LIN {X 0,Y 302.598,Z 692.488,A -85,B 0,C 180,E1 10469.522,E2 10469.522} C_VEL
LIN {X 0,Y 304.886,Z 667.23,A -85,B 0,C 180,E1 10468.838,E2 10468.838} C_VEL
LIN {X 0,Y 315.43,Z 536.888,A -85,B 0,C 180,E1 10466.199,E2 10466.199} C_VEL
LIN {X 0,Y 309.663,Z 526.865,A -85,B 0,C 180,E1 10462.898,E2 10462.898} C_VEL
LIN {X 0,Y 304.796,Z 519.088,A -85,B 0,C 180,E1 10459.549,E2 10459.549} C_VEL
LIN {X 0,Y 301.581,Z 514.357,A -85,B 0,C 180,E1 10456.864,E2 10456.864} C_VEL
LIN {X 0,Y 300.41,Z 512.771,A -85,B 0,C 180,E1 10455.75,E2 10455.75} C_VEL
LIN {X 0,Y 298.97,Z 511.709,A -85,B 0,C 180,E1 10454.313,E2 10454.313} C_VEL
LIN {X 0,Y 296.741,Z 512.653,A -85,B 0,C 180,E1 10451.996,E2 10451.996} C_VEL
LIN {X 0,Y 294.887,Z 513.836,A -85,B 0,C 180,E1 10449.52,E2 10449.52} C_VEL
LIN {X 0,Y 294.603,Z 513.741,A -85,B 0,C 180,E1 10448.976,E2 10448.976} C_VEL
LIN {X 0,Y 293.288,Z 512.887,A -85,B 0,C 180,E1 10444.302,E2 10444.302} C_VEL
LIN {X 0,Y 293.492,Z 513.574,A -85,B 0,C 180,E1 10440.391,E2 10440.391} C_VEL
LIN {X 0,Y 295.393,Z 518.005,A -85,B 0,C 180,E1 10435.341,E2 10435.341} C_VEL
LIN {X 0,Y 297.878,Z 523.02,A -85,B 0,C 180,E1 10431.799,E2 10431.799} C_VEL
LIN {X 0,Y 299.981,Z 527.143,A -85,B 0,C 180,E1 10429.534,E2 10429.534} C_VEL
LIN {X 0,Y 303.204,Z 533.381,A -85,B 0,C 180,E1 10426.703,E2 10426.703} C_VEL
LIN {X 0,Y 307.026,Z 541.211,A -85,B 0,C 180,E1 10423.882,E2 10423.882} C_VEL
LIN {X 0,Y 311.626,Z 551.031,A -85,B 0,C 180,E1 10420.995,E2 10420.995} C_VEL
LIN {X 0,Y 312.497,Z 553.268,A -85,B 0,C 180,E1 10420.473,E2 10420.473} C_VEL
LIN {X 0,Y 297.53,Z 720.46,A -85,B 0,C 180,E1 10416.945,E2 10416.945} C_VEL
LIN {X 0,Y 293.952,Z 742.565,A -85,B 0,C 180,E1 10416.298,E2 10416.298} C_VEL
LIN {X 0,Y 288.986,Z 764.025,A -85,B 0,C 180,E1 10415.487,E2 10415.487} C_VEL
LIN {X 0,Y 282.983,Z 784.23,A -85,B 0,C 180,E1 10414.512,E2 10414.512} C_VEL
LIN {X 0,Y 275.952,Z 803.851,A -85,B 0,C 180,E1 10413.261,E2 10413.261} C_VEL
LIN {X 0,Y 268.029,Z 822.907,A -85,B 0,C 180,E1 10411.679,E2 10411.679} C_VEL
LIN {X 0,Y 258.872,Z 842.398,A -85,B 0,C 180,E1 10409.605,E2 10409.605} C_VEL
LIN {X 0,Y 249.5,Z 860.393,A -85,B 0,C 180,E1 10407.16,E2 10407.16} C_VEL
LIN {X 0,Y 239.675,Z 877.621,A -85,B 0,C 180,E1 10404.172,E2 10404.172} C_VEL
LIN {X 0,Y 230.079,Z 893.458,A -85,B 0,C 180,E1 10400.667,E2 10400.667} C_VEL
LIN {X 0,Y 220.636,Z 908.459,A -85,B 0,C 180,E1 10396.464,E2 10396.464} C_VEL
LIN {X 0,Y 212.557,Z 921.328,A -85,B 0,C 180,E1 10391.906,E2 10391.906} C_VEL
LIN {X 0,Y 205.237,Z 933.456,A -85,B 0,C 180,E1 10386.463,E2 10386.463} C_VEL
LIN {X 0,Y 199.633,Z 943.745,A -85,B 0,C 180,E1 10380.521,E2 10380.521} C_VEL
LIN {X 0,Y 196.02,Z 952.022,A -85,B 0,C 180,E1 10374.402,E2 10374.402} C_VEL
LIN {X 0,Y 194.187,Z 958.687,A -85,B 0,C 180,E1 10367.994,E2 10367.994} C_VEL
LIN {X 0,Y 193.926,Z 963.068,A -85,B 0,C 180,E1 10362.204,E2 10362.204} C_VEL
LIN {X 0,Y 194.453,Z 965.803,A -85,B 0,C 180,E1 10356.792,E2 10356.792} C_VEL
LIN {X 0,Y 194.986,Z 966.923,A -85,B 0,C 180,E1 10352.352,E2 10352.352} C_VEL
LIN {X 0,Y 195.041,Z 967.009,A -85,B 0,C 180,E1 10348.457,E2 10348.457} C_VEL
LIN {X 0,Y 194.615,Z 966.173,A -85,B 0,C 180,E1 10344.4,E2 10344.4} C_VEL
LIN {X 0,Y 194.022,Z 963.972,A -85,B 0,C 180,E1 10339.311,E2 10339.311} C_VEL
LIN {X 0,Y 194.046,Z 959.689,A -85,B 0,C 180,E1 10333.232,E2 10333.232} C_VEL
LIN {X 0,Y 195.44,Z 953.707,A -85,B 0,C 180,E1 10327.051,E2 10327.051} C_VEL
LIN {X 0,Y 198.684,Z 945.671,A -85,B 0,C 180,E1 10320.786,E2 10320.786} C_VEL
LIN {X 0,Y 203.684,Z 936.028,A -85,B 0,C 180,E1 10314.952,E2 10314.952} C_VEL
LIN {X 0,Y 210.542,Z 924.446,A -85,B 0,C 180,E1 10309.419,E2 10309.419} C_VEL
LIN {X 0,Y 218.263,Z 912.191,A -85,B 0,C 180,E1 10304.768,E2 10304.768} C_VEL
LIN {X 0,Y 227.319,Z 897.792,A -85,B 0,C 180,E1 10300.461,E2 10300.461} C_VEL
LIN {X 0,Y 236.604,Z 882.589,A -85,B 0,C 180,E1 10296.875,E2 10296.875} C_VEL
LIN {X 0,Y 246.735,Z 865.128,A -85,B 0,C 180,E1 10293.627,E2 10293.627} C_VEL
LIN {X 0,Y 256.161,Z 847.562,A -85,B 0,C 180,E1 10291.056,E2 10291.056} C_VEL
LIN {X 0,Y 265.436,Z 828.501,A -85,B 0,C 180,E1 10288.873,E2 10288.873} C_VEL
LIN {X 0,Y 273.54,Z 809.538,A -85,B 0,C 180,E1 10287.187,E2 10287.187} C_VEL
LIN {X 0,Y 280.979,Z 789.632,A -85,B 0,C 180,E1 10285.817,E2 10285.817} C_VEL
LIN {X 0,Y 287.475,Z 769.122,A -85,B 0,C 180,E1 10284.747,E2 10284.747} C_VEL
LIN {X 0,Y 293.011,Z 746.686,A -85,B 0,C 180,E1 10283.853,E2 10283.853} C_VEL
LIN {X 0,Y 296.814,Z 724.483,A -85,B 0,C 180,E1 10283.178,E2 10283.178} C_VEL
LIN {X 0,Y 299.999,Z 692.914,A -85,B 0,C 180,E1 10282.46,E2 10282.46} C_VEL
LIN {X 0,Y 312.304,Z 552.77,A -85,B 0,C 180,E1 10279.497,E2 10279.497} C_VEL
LIN {X 0,Y 307.54,Z 542.415,A -85,B 0,C 180,E1 10276.576,E2 10276.576} C_VEL
LIN {X 0,Y 303.48,Z 534.184,A -85,B 0,C 180,E1 10273.673,E2 10273.673} C_VEL
LIN {X 0,Y 300.18,Z 527.74,A -85,B 0,C 180,E1 10270.847,E2 10270.847} C_VEL
LIN {X 0,Y 298.085,Z 523.643,A -85,B 0,C 180,E1 10268.681,E2 10268.681} C_VEL
LIN {X 0,Y 296.396,Z 520.441,A -85,B 0,C 180,E1 10266.586,E2 10266.586} C_VEL
LIN {X 0,Y 294.859,Z 517.125,A -85,B 0,C 180,E1 10264.083,E2 10264.083} C_VEL
LIN {X 0,Y 293.192,Z 513.211,A -85,B 0,C 180,E1 10259.218,E2 10259.218} C_VEL
LIN {X 0,Y 293.326,Z 512.761,A -85,B 0,C 180,E1 10253.934,E2 10253.934} C_VEL
LIN {X 0,Y 294.723,Z 513.985,A -85,B 0,C 180,E1 10250.233,E2 10250.233} C_VEL
LIN {X 0,Y 298.119,Z 518.939,A -85,B 0,C 180,E1 10245.332,E2 10245.332} C_VEL
LIN {X 0,Y 301.263,Z 523.806,A -85,B 0,C 180,E1 10242.221,E2 10242.221} C_VEL
LIN {X 0,Y 304.449,Z 528.849,A -85,B 0,C 180,E1 10239.677,E2 10239.677} C_VEL
LIN {X 0,Y 309.247,Z 536.938,A -85,B 0,C 180,E1 10236.465,E2 10236.465} C_VEL
LIN {X 0,Y 311.824,Z 541.761,A -85,B 0,C 180,E1 10234.936,E2 10234.936} C_VEL
LIN {X 0,Y 300.184,Z 680.951,A -85,B 0,C 180,E1 10232.1,E2 10232.1} C_VEL
LIN {X 0,Y 297.715,Z 701.831,A -85,B 0,C 180,E1 10231.431,E2 10231.431} C_VEL
LIN {X 0,Y 293.977,Z 722.266,A -85,B 0,C 180,E1 10230.528,E2 10230.528} C_VEL
LIN {X 0,Y 289.19,Z 741.453,A -85,B 0,C 180,E1 10229.407,E2 10229.407} C_VEL
LIN {X 0,Y 283.05,Z 761.038,A -85,B 0,C 180,E1 10227.961,E2 10227.961} C_VEL
LIN {X 0,Y 275.997,Z 779.593,A -85,B 0,C 180,E1 10226.234,E2 10226.234} C_VEL
LIN {X 0,Y 268.131,Z 797.188,A -85,B 0,C 180,E1 10224.19,E2 10224.19} C_VEL
LIN {X 0,Y 259.42,Z 813.987,A -85,B 0,C 180,E1 10221.736,E2 10221.736} C_VEL
LIN {X 0,Y 250.527,Z 829.117,A -85,B 0,C 180,E1 10218.957,E2 10218.957} C_VEL
LIN {X 0,Y 241.45,Z 843.036,A -85,B 0,C 180,E1 10215.751,E2 10215.751} C_VEL
LIN {X 0,Y 232.571,Z 855.538,A -85,B 0,C 180,E1 10212.112,E2 10212.112} C_VEL
LIN {X 0,Y 224.082,Z 866.647,A -85,B 0,C 180,E1 10208.001,E2 10208.001} C_VEL
LIN {X 0,Y 215.89,Z 876.71,A -85,B 0,C 180,E1 10203.122,E2 10203.122} C_VEL
LIN {X 0,Y 209.066,Z 884.767,A -85,B 0,C 180,E1 10197.945,E2 10197.945} C_VEL
LIN {X 0,Y 203.512,Z 891.329,A -85,B 0,C 180,E1 10192.225,E2 10192.225} C_VEL
LIN {X 0,Y 199.383,Z 896.318,A -85,B 0,C 180,E1 10186.008,E2 10186.008} C_VEL
LIN {X 0,Y 197.027,Z 899.441,A -85,B 0,C 180,E1 10179.934,E2 10179.934} C_VEL
LIN {X 0,Y 195.894,Z 901.059,A -85,B 0,C 180,E1 10173.803,E2 10173.803} C_VEL
LIN {X 0,Y 195.752,Z 901.224,A -85,B 0,C 180,E1 10167.95,E2 10167.95} C_VEL
LIN {X 0,Y 196.557,Z 900.078,A -85,B 0,C 180,E1 10161.811,E2 10161.811} C_VEL
LIN {X 0,Y 198.545,Z 897.495,A -85,B 0,C 180,E1 10155.715,E2 10155.715} C_VEL
LIN {X 0,Y 202.162,Z 893.041,A -85,B 0,C 180,E1 10149.443,E2 10149.443} C_VEL
LIN {X 0,Y 207.241,Z 887,A -85,B 0,C 180,E1 10143.651,E2 10143.651} C_VEL
LIN {X 0,Y 213.604,Z 879.489,A -85,B 0,C 180,E1 10138.384,E2 10138.384} C_VEL
LIN {X 0,Y 221.371,Z 870.076,A -85,B 0,C 180,E1 10133.405,E2 10133.405} C_VEL
LIN {X 0,Y 229.529,Z 859.758,A -85,B 0,C 180,E1 10129.204,E2 10129.204} C_VEL
LIN {X 0,Y 238.649,Z 847.341,A -85,B 0,C 180,E1 10125.267,E2 10125.267} C_VEL
LIN {X 0,Y 247.506,Z 834.121,A -85,B 0,C 180,E1 10121.991,E2 10121.991} C_VEL
LIN {X 0,Y 256.534,Z 819.275,A -85,B 0,C 180,E1 10119.053,E2 10119.053} C_VEL
LIN {X 0,Y 265.427,Z 802.853,A -85,B 0,C 180,E1 10116.469,E2 10116.469} C_VEL
LIN {X 0,Y 273.225,Z 786.497,A -85,B 0,C 180,E1 10114.397,E2 10114.397} C_VEL
LIN {X 0,Y 280.677,Z 768.155,A -85,B 0,C 180,E1 10112.542,E2 10112.542} C_VEL
LIN {X 0,Y 286.961,Z 749.583,A -85,B 0,C 180,E1 10111.043,E2 10111.043} C_VEL
LIN {X 0,Y 292.498,Z 729.301,A -85,B 0,C 180,E1 10109.752,E2 10109.752} C_VEL
LIN {X 0,Y 296.633,Z 709.476,A -85,B 0,C 180,E1 10108.775,E2 10108.775} C_VEL
LIN {X 0,Y 299.604,Z 688.99,A -85,B 0,C 180,E1 10108.026,E2 10108.026} C_VEL
LIN {X 0,Y 302.276,Z 657.024,A -85,B 0,C 180,E1 10107.247,E2 10107.247} C_VEL
LIN {X 0,Y 311.954,Z 541.598,A -85,B 0,C 180,E1 10104.928,E2 10104.928} C_VEL
LIN {X 0,Y 306.944,Z 532.838,A -85,B 0,C 180,E1 10101.85,E2 10101.85} C_VEL
LIN {X 0,Y 302.881,Z 526.177,A -85,B 0,C 180,E1 10098.876,E2 10098.876} C_VEL
LIN {X 0,Y 300.118,Z 521.934,A -85,B 0,C 180,E1 10096.451,E2 10096.451} C_VEL
LIN {X 0,Y 297.658,Z 518.183,A -85,B 0,C 180,E1 10093.798,E2 10093.798} C_VEL
LIN {X 0,Y 294.603,Z 513.741,A -85,B 0,C 180,E1 10088.976,E2 10088.976} C_VEL
LIN {X 0,Y 293.866,Z 514.281,A -85,B 0,C 180,E1 10087.476,E2 10087.476} C_VEL
LIN {X 0,Y 292.602,Z 518.683,A -85,B 0,C 180,E1 10084.538,E2 10084.538} C_VEL
LIN {X 0,Y 292.268,Z 520.81,A -85,B 0,C 180,E1 10082.715,E2 10082.715} C_VEL
LIN {X 0,Y 292.277,Z 521.017,A -85,B 0,C 180,E1 10082.167,E2 10082.167} C_VEL
LIN {X 0,Y 292.498,Z 521.631,A -85,B 0,C 180,E1 10080.392,E2 10080.392} C_VEL
LIN {X 0,Y 294.224,Z 525.821,A -85,B 0,C 180,E1 10075.615,E2 10075.615} C_VEL
LIN {X 0,Y 296.463,Z 530.543,A -85,B 0,C 180,E1 10072.247,E2 10072.247} C_VEL
LIN {X 0,Y 298.569,Z 534.867,A -85,B 0,C 180,E1 10069.874,E2 10069.874} C_VEL
LIN {X 0,Y 301.629,Z 541.097,A -85,B 0,C 180,E1 10067.071,E2 10067.071} C_VEL
LIN {X 0,Y 305.547,Z 549.403,A -85,B 0,C 180,E1 10064.094,E2 10064.094} C_VEL
LIN {X 0,Y 309.101,Z 557.525,A -85,B 0,C 180,E1 10061.755,E2 10061.755} C_VEL
LIN {X 0,Y 294.187,Z 719.498,A -85,B 0,C 180,E1 10058.368,E2 10058.368} C_VEL
LIN {X 0,Y 290.514,Z 741.649,A -85,B 0,C 180,E1 10057.73,E2 10057.73} C_VEL
LIN {X 0,Y 285.497,Z 762.884,A -85,B 0,C 180,E1 10056.943,E2 10056.943} C_VEL
LIN {X 0,Y 279.162,Z 783.671,A -85,B 0,C 180,E1 10055.957,E2 10055.957} C_VEL
LIN {X 0,Y 271.966,Z 803.225,A -85,B 0,C 180,E1 10054.732,E2 10054.732} C_VEL
LIN {X 0,Y 263.871,Z 822.089,A -85,B 0,C 180,E1 10053.185,E2 10053.185} C_VEL
LIN {X 0,Y 254.528,Z 841.356,A -85,B 0,C 180,E1 10051.156,E2 10051.156} C_VEL
LIN {X 0,Y 245.066,Z 858.936,A -85,B 0,C 180,E1 10048.792,E2 10048.792} C_VEL
LIN {X 0,Y 234.724,Z 876.375,A -85,B 0,C 180,E1 10045.787,E2 10045.787} C_VEL
LIN {X 0,Y 224.834,Z 891.994,A -85,B 0,C 180,E1 10042.328,E2 10042.328} C_VEL
LIN {X 0,Y 214.92,Z 907.001,A -85,B 0,C 180,E1 10038.099,E2 10038.099} C_VEL
LIN {X 0,Y 206.335,Z 919.888,A -85,B 0,C 180,E1 10033.476,E2 10033.476} C_VEL
LIN {X 0,Y 198.503,Z 932.02,A -85,B 0,C 180,E1 10027.913,E2 10027.913} C_VEL
LIN {X 0,Y 192.57,Z 942.042,A -85,B 0,C 180,E1 10021.976,E2 10021.976} C_VEL
LIN {X 0,Y 188.436,Z 950.612,A -85,B 0,C 180,E1 10015.453,E2 10015.453} C_VEL
LIN {X 0,Y 186.396,Z 957.036,A -85,B 0,C 180,E1 10009.099,E2 10009.099} C_VEL
LIN {X 0,Y 185.959,Z 961.492,A -85,B 0,C 180,E1 10003.051,E2 10003.051} C_VEL
LIN {X 0,Y 186.495,Z 964.454,A -85,B 0,C 180,E1 9997.084,E2 9997.084} C_VEL
LIN {X 0,Y 187.084,Z 965.592,A -85,B 0,C 180,E1 9992.451,E2 9992.451} C_VEL
LIN {X 0,Y 187.15,Z 965.687,A -85,B 0,C 180,E1 9988.471,E2 9988.471} C_VEL
LIN {X 0,Y 186.667,Z 964.828,A -85,B 0,C 180,E1 9984.161,E2 9984.161} C_VEL
LIN {X 0,Y 186.028,Z 962.452,A -85,B 0,C 180,E1 9978.532,E2 9978.532} C_VEL
LIN {X 0,Y 186.163,Z 958.299,A -85,B 0,C 180,E1 9972.499,E2 9972.499} C_VEL
LIN {X 0,Y 187.758,Z 952.379,A -85,B 0,C 180,E1 9966.13,E2 9966.13} C_VEL
LIN {X 0,Y 191.412,Z 944.212,A -85,B 0,C 180,E1 9959.528,E2 9959.528} C_VEL
LIN {X 0,Y 196.833,Z 934.597,A -85,B 0,C 180,E1 9953.541,E2 9953.541} C_VEL
LIN {X 0,Y 204.197,Z 923.004,A -85,B 0,C 180,E1 9947.876,E2 9947.876} C_VEL
LIN {X 0,Y 212.762,Z 910.147,A -85,B 0,C 180,E1 9942.953,E2 9942.953} C_VEL
LIN {X 0,Y 222.519,Z 895.499,A -85,B 0,C 180,E1 9938.579,E2 9938.579} C_VEL
LIN {X 0,Y 232.777,Z 879.347,A -85,B 0,C 180,E1 9934.839,E2 9934.839} C_VEL
LIN {X 0,Y 242.831,Z 862.546,A -85,B 0,C 180,E1 9931.805,E2 9931.805} C_VEL
LIN {X 0,Y 253.056,Z 843.933,A -85,B 0,C 180,E1 9929.179,E2 9929.179} C_VEL
LIN {X 0,Y 262.303,Z 825.275,A -85,B 0,C 180,E1 9927.131,E2 9927.131} C_VEL
LIN {X 0,Y 270.768,Z 805.846,A -85,B 0,C 180,E1 9925.477,E2 9925.477} C_VEL
LIN {X 0,Y 277.967,Z 786.635,A -85,B 0,C 180,E1 9924.227,E2 9924.227} C_VEL
LIN {X 0,Y 284.865,Z 764.64,A -85,B 0,C 180,E1 9923.147,E2 9923.147} C_VEL
LIN {X 0,Y 290.09,Z 743.05,A -85,B 0,C 180,E1 9922.329,E2 9922.329} C_VEL
LIN {X 0,Y 293.893,Z 720.546,A -85,B 0,C 180,E1 9921.672,E2 9921.672} C_VEL
LIN {X 0,Y 300.961,Z 644.8,A -85,B 0,C 180,E1 9920.048,E2 9920.048} C_VEL
LIN {X 0,Y 308.94,Z 557.28,A -85,B 0,C 180,E1 9918.247,E2 9918.247} C_VEL
LIN {X 0,Y 304.478,Z 547.365,A -85,B 0,C 180,E1 9915.279,E2 9915.279} C_VEL
LIN {X 0,Y 300.744,Z 539.393,A -85,B 0,C 180,E1 9912.333,E2 9912.333} C_VEL
LIN {X 0,Y 296.979,Z 531.794,A -85,B 0,C 180,E1 9908.616,E2 9908.616} C_VEL
LIN {X 0,Y 295.114,Z 528.114,A -85,B 0,C 180,E1 9906.224,E2 9906.224} C_VEL
LIN {X 0,Y 293.656,Z 524.851,A -85,B 0,C 180,E1 9903.709,E2 9903.709} C_VEL
LIN {X 0,Y 292.181,Z 521.109,A -85,B 0,C 180,E1 9899.019,E2 9899.019} C_VEL
LIN {X 0,Y 292.36,Z 520.705,A -85,B 0,C 180,E1 9893.914,E2 9893.914} C_VEL
LIN {X 0,Y 293.663,Z 521.892,A -85,B 0,C 180,E1 9890.396,E2 9890.396} C_VEL
LIN {X 0,Y 296.898,Z 526.806,A -85,B 0,C 180,E1 9885.569,E2 9885.569} C_VEL
LIN {X 0,Y 299.771,Z 531.371,A -85,B 0,C 180,E1 9882.631,E2 9882.631} C_VEL
LIN {X 0,Y 303.041,Z 536.731,A -85,B 0,C 180,E1 9879.931,E2 9879.931} C_VEL
LIN {X 0,Y 307.61,Z 544.732,A -85,B 0,C 180,E1 9876.789,E2 9876.789} C_VEL
LIN {X 0,Y 308.491,Z 546.693,A -85,B 0,C 180,E1 9876.221,E2 9876.221} C_VEL
LIN {X 0,Y 296.837,Z 681.695,A -85,B 0,C 180,E1 9873.487,E2 9873.487} C_VEL
LIN {X 0,Y 294.299,Z 702.606,A -85,B 0,C 180,E1 9872.823,E2 9872.823} C_VEL
LIN {X 0,Y 290.385,Z 723.397,A -85,B 0,C 180,E1 9871.912,E2 9871.912} C_VEL
LIN {X 0,Y 285.285,Z 743.188,A -85,B 0,C 180,E1 9870.761,E2 9870.761} C_VEL
LIN {X 0,Y 279.317,Z 761.66,A -85,B 0,C 180,E1 9869.408,E2 9869.408} C_VEL
LIN {X 0,Y 272.399,Z 779.534,A -85,B 0,C 180,E1 9867.776,E2 9867.776} C_VEL
LIN {X 0,Y 264.312,Z 797.22,A -85,B 0,C 180,E1 9865.761,E2 9865.761} C_VEL
LIN {X 0,Y 255.739,Z 813.37,A -85,B 0,C 180,E1 9863.451,E2 9863.451} C_VEL
LIN {X 0,Y 246.635,Z 828.587,A -85,B 0,C 180,E1 9860.734,E2 9860.734} C_VEL
LIN {X 0,Y 237.143,Z 842.817,A -85,B 0,C 180,E1 9857.541,E2 9857.541} C_VEL
LIN {X 0,Y 227.812,Z 855.586,A -85,B 0,C 180,E1 9853.897,E2 9853.897} C_VEL
LIN {X 0,Y 218.353,Z 867.424,A -85,B 0,C 180,E1 9849.525,E2 9849.525} C_VEL
LIN {X 0,Y 210.075,Z 877.112,A -85,B 0,C 180,E1 9844.825,E2 9844.825} C_VEL
LIN {X 0,Y 202.734,Z 885.373,A -85,B 0,C 180,E1 9839.546,E2 9839.546} C_VEL
LIN {X 0,Y 196.678,Z 892.127,A -85,B 0,C 180,E1 9833.676,E2 9833.676} C_VEL
LIN {X 0,Y 192.273,Z 897.113,A -85,B 0,C 180,E1 9827.551,E2 9827.551} C_VEL
LIN {X 0,Y 189.518,Z 900.442,A -85,B 0,C 180,E1 9821.254,E2 9821.254} C_VEL
LIN {X 0,Y 188.111,Z 902.212,A -85,B 0,C 180,E1 9814.877,E2 9814.877} C_VEL
LIN {X 0,Y 187.845,Z 902.59,A -85,B 0,C 180,E1 9808.474,E2 9808.474} C_VEL
LIN {X 0,Y 188.548,Z 901.703,A -85,B 0,C 180,E1 9802.381,E2 9802.381} C_VEL
LIN {X 0,Y 190.485,Z 899.267,A -85,B 0,C 180,E1 9796.028,E2 9796.028} C_VEL
LIN {X 0,Y 193.901,Z 895.276,A -85,B 0,C 180,E1 9789.789,E2 9789.789} C_VEL
LIN {X 0,Y 199.276,Z 889.293,A -85,B 0,C 180,E1 9783.479,E2 9783.479} C_VEL
LIN {X 0,Y 205.782,Z 882.091,A -85,B 0,C 180,E1 9778.023,E2 9778.023} C_VEL
LIN {X 0,Y 213.749,Z 873.014,A -85,B 0,C 180,E1 9772.888,E2 9772.888} C_VEL
LIN {X 0,Y 222.592,Z 862.366,A -85,B 0,C 180,E1 9768.337,E2 9768.337} C_VEL
LIN {X 0,Y 231.436,Z 850.873,A -85,B 0,C 180,E1 9764.538,E2 9764.538} C_VEL
LIN {X 0,Y 241.102,Z 837.252,A -85,B 0,C 180,E1 9761.001,E2 9761.001} C_VEL
LIN {X 0,Y 250.542,Z 822.535,A -85,B 0,C 180,E1 9757.99,E2 9757.99} C_VEL
LIN {X 0,Y 259.518,Z 806.852,A -85,B 0,C 180,E1 9755.433,E2 9755.433} C_VEL
LIN {X 0,Y 267.837,Z 790.127,A -85,B 0,C 180,E1 9753.265,E2 9753.265} C_VEL
LIN {X 0,Y 275.373,Z 772.583,A -85,B 0,C 180,E1 9751.439,E2 9751.439} C_VEL
LIN {X 0,Y 282.351,Z 753.244,A -85,B 0,C 180,E1 9749.829,E2 9749.829} C_VEL
LIN {X 0,Y 287.994,Z 734.014,A -85,B 0,C 180,E1 9748.563,E2 9748.563} C_VEL
LIN {X 0,Y 292.536,Z 713.8,A -85,B 0,C 180,E1 9747.531,E2 9747.531} C_VEL
LIN {X 0,Y 295.735,Z 693.527,A -85,B 0,C 180,E1 9746.759,E2 9746.759} C_VEL
LIN {X 0,Y 298.213,Z 667.402,A -85,B 0,C 180,E1 9746.068,E2 9746.068} C_VEL
LIN {X 0,Y 308.621,Z 546.478,A -85,B 0,C 180,E1 9743.636,E2 9743.636} C_VEL
LIN {X 0,Y 303.836,Z 537.808,A -85,B 0,C 180,E1 9740.416,E2 9740.416} C_VEL
LIN {X 0,Y 300.367,Z 532.238,A -85,B 0,C 180,E1 9737.633,E2 9737.633} C_VEL
LIN {X 0,Y 298.478,Z 529.25,A -85,B 0,C 180,E1 9735.844,E2 9735.844} C_VEL
LIN {X 0,Y 296.384,Z 525.912,A -85,B 0,C 180,E1 9733.461,E2 9733.461} C_VEL
LIN {X 0,Y 293.465,Z 521.568,A -85,B 0,C 180,E1 9728.622,E2 9728.622} C_VEL
LIN {X 0,Y 292.296,Z 520.836,A -85,B 0,C 180,E1 9724.12,E2 9724.12} C_VEL
LIN {X 0,Y 292.277,Z 521.017,A -85,B 0,C 180,E1 9722.167,E2 9722.167} C_VEL
LIN {X 0,Y 292.332,Z 522.09,A -85,B 0,C 180,E1 9720.888,E2 9720.888} C_VEL
LIN {X 0,Y 292.38,Z 525.919,A -85,B 0,C 180,E1 9719.074,E2 9719.074} C_VEL
LIN {X 0,Y 292.897,Z 532.914,A -85,B 0,C 180,E1 9716.288,E2 9716.288} C_VEL
LIN {X 0,Y 293.177,Z 533.967,A -85,B 0,C 180,E1 9715.66,E2 9715.66} C_VEL
LIN {X 0,Y 295.213,Z 538.391,A -85,B 0,C 180,E1 9712.508,E2 9712.508} C_VEL
LIN {X 0,Y 297.257,Z 542.775,A -85,B 0,C 180,E1 9710.123,E2 9710.123} C_VEL
LIN {X 0,Y 300.507,Z 549.737,A -85,B 0,C 180,E1 9707.071,E2 9707.071} C_VEL
LIN {X 0,Y 304.375,Z 558.476,A -85,B 0,C 180,E1 9704.081,E2 9704.081} C_VEL
LIN {X 0,Y 305.827,Z 562.147,A -85,B 0,C 180,E1 9703.058,E2 9703.058} C_VEL
LIN {X 0,Y 291.029,Z 718.539,A -85,B 0,C 180,E1 9699.824,E2 9699.824} C_VEL
LIN {X 0,Y 287.259,Z 740.757,A -85,B 0,C 180,E1 9699.195,E2 9699.195} C_VEL
LIN {X 0,Y 281.987,Z 762.493,A -85,B 0,C 180,E1 9698.403,E2 9698.403} C_VEL
LIN {X 0,Y 275.523,Z 783.116,A -85,B 0,C 180,E1 9697.441,E2 9697.441} C_VEL
LIN {X 0,Y 268.022,Z 802.964,A -85,B 0,C 180,E1 9696.221,E2 9696.221} C_VEL
LIN {X 0,Y 259.474,Z 822.195,A -85,B 0,C 180,E1 9694.654,E2 9694.654} C_VEL
LIN {X 0,Y 249.883,Z 841.231,A -85,B 0,C 180,E1 9692.65,E2 9692.65} C_VEL
LIN {X 0,Y 240.101,Z 858.69,A -85,B 0,C 180,E1 9690.294,E2 9690.294} C_VEL
LIN {X 0,Y 229.352,Z 876.133,A -85,B 0,C 180,E1 9687.278,E2 9687.278} C_VEL
LIN {X 0,Y 219.181,Z 891.444,A -85,B 0,C 180,E1 9683.84,E2 9683.84} C_VEL
LIN {X 0,Y 209.379,Z 905.552,A -85,B 0,C 180,E1 9679.818,E2 9679.818} C_VEL
LIN {X 0,Y 200.281,Z 918.45,A -85,B 0,C 180,E1 9675.141,E2 9675.141} C_VEL
LIN {X 0,Y 191.905,Z 930.585,A -85,B 0,C 180,E1 9669.464,E2 9669.464} C_VEL
LIN {X 0,Y 185.43,Z 940.692,A -85,B 0,C 180,E1 9663.305,E2 9663.305} C_VEL
LIN {X 0,Y 180.91,Z 949.2,A -85,B 0,C 180,E1 9656.593,E2 9656.593} C_VEL
LIN {X 0,Y 178.563,Z 955.748,A -85,B 0,C 180,E1 9649.831,E2 9649.831} C_VEL
LIN {X 0,Y 177.997,Z 960.114,A -85,B 0,C 180,E1 9643.646,E2 9643.646} C_VEL
LIN {X 0,Y 178.511,Z 963.064,A -85,B 0,C 180,E1 9637.527,E2 9637.527} C_VEL
LIN {X 0,Y 179.169,Z 964.246,A -85,B 0,C 180,E1 9632.683,E2 9632.683} C_VEL
LIN {X 0,Y 179.271,Z 964.388,A -85,B 0,C 180,E1 9628.723,E2 9628.723} C_VEL
LIN {X 0,Y 178.801,Z 963.653,A -85,B 0,C 180,E1 9624.482,E2 9624.482} C_VEL
LIN {X 0,Y 178.151,Z 961.62,A -85,B 0,C 180,E1 9619.16,E2 9619.16} C_VEL
LIN {X 0,Y 178.215,Z 957.421,A -85,B 0,C 180,E1 9612.367,E2 9612.367} C_VEL
LIN {X 0,Y 179.882,Z 951.664,A -85,B 0,C 180,E1 9605.716,E2 9605.716} C_VEL
LIN {X 0,Y 183.706,Z 943.658,A -85,B 0,C 180,E1 9598.87,E2 9598.87} C_VEL
LIN {X 0,Y 189.42,Z 934.208,A -85,B 0,C 180,E1 9592.631,E2 9592.631} C_VEL
LIN {X 0,Y 196.755,Z 923.386,A -85,B 0,C 180,E1 9587.034,E2 9587.034} C_VEL
LIN {X 0,Y 205.663,Z 910.752,A -85,B 0,C 180,E1 9581.949,E2 9581.949} C_VEL
LIN {X 0,Y 214.999,Z 897.384,A -85,B 0,C 180,E1 9577.769,E2 9577.769} C_VEL
LIN {X 0,Y 225.742,Z 881.443,A -85,B 0,C 180,E1 9573.863,E2 9573.863} C_VEL
LIN {X 0,Y 235.633,Z 865.94,A -85,B 0,C 180,E1 9570.892,E2 9570.892} C_VEL
LIN {X 0,Y 246.153,Z 847.895,A -85,B 0,C 180,E1 9568.196,E2 9568.196} C_VEL
LIN {X 0,Y 255.546,Z 829.98,A -85,B 0,C 180,E1 9566.124,E2 9566.124} C_VEL
LIN {X 0,Y 264.969,Z 809.695,A -85,B 0,C 180,E1 9564.303,E2 9564.303} C_VEL
LIN {X 0,Y 273.024,Z 789.643,A -85,B 0,C 180,E1 9562.938,E2 9562.938} C_VEL
LIN {X 0,Y 280.09,Z 768.679,A -85,B 0,C 180,E1 9561.869,E2 9561.869} C_VEL
LIN {X 0,Y 285.821,Z 746.711,A -85,B 0,C 180,E1 9561.017,E2 9561.017} C_VEL
LIN {X 0,Y 289.931,Z 724.744,A -85,B 0,C 180,E1 9560.354,E2 9560.354} C_VEL
LIN {X 0,Y 293.177,Z 695.947,A -85,B 0,C 180,E1 9559.697,E2 9559.697} C_VEL
LIN {X 0,Y 305.654,Z 561.652,A -85,B 0,C 180,E1 9556.926,E2 9556.926} C_VEL
LIN {X 0,Y 300.89,Z 550.718,A -85,B 0,C 180,E1 9553.401,E2 9553.401} C_VEL
LIN {X 0,Y 297.431,Z 543.352,A -85,B 0,C 180,E1 9550.263,E2 9550.263} C_VEL
LIN {X 0,Y 295.087,Z 538.367,A -85,B 0,C 180,E1 9547.593,E2 9547.593} C_VEL
LIN {X 0,Y 292.664,Z 532.867,A -85,B 0,C 180,E1 9543.721,E2 9543.721} C_VEL
LIN {X 0,Y 291.173,Z 529.007,A -85,B 0,C 180,E1 9538.819,E2 9538.819} C_VEL
LIN {X 0,Y 291.439,Z 528.681,A -85,B 0,C 180,E1 9533.697,E2 9533.697} C_VEL
LIN {X 0,Y 292.605,Z 529.799,A -85,B 0,C 180,E1 9530.559,E2 9530.559} C_VEL
LIN {X 0,Y 295.605,Z 534.517,A -85,B 0,C 180,E1 9525.904,E2 9525.904} C_VEL
LIN {X 0,Y 298.393,Z 539.115,A -85,B 0,C 180,E1 9522.95,E2 9522.95} C_VEL
LIN {X 0,Y 301.461,Z 544.306,A -85,B 0,C 180,E1 9520.327,E2 9520.327} C_VEL
LIN {X 0,Y 305.338,Z 551.347,A -85,B 0,C 180,E1 9517.539,E2 9517.539} C_VEL
LIN {X 0,Y 293.668,Z 682.444,A -85,B 0,C 180,E1 9514.905,E2 9514.905} C_VEL
LIN {X 0,Y 291.061,Z 703.38,A -85,B 0,C 180,E1 9514.247,E2 9514.247} C_VEL
LIN {X 0,Y 286.966,Z 724.525,A -85,B 0,C 180,E1 9513.33,E2 9513.33} C_VEL
LIN {X 0,Y 281.902,Z 743.673,A -85,B 0,C 180,E1 9512.231,E2 9512.231} C_VEL
LIN {X 0,Y 275.407,Z 763.253,A -85,B 0,C 180,E1 9510.812,E2 9510.812} C_VEL
LIN {X 0,Y 267.936,Z 781.821,A -85,B 0,C 180,E1 9509.114,E2 9509.114} C_VEL
LIN {X 0,Y 259.65,Z 799.313,A -85,B 0,C 180,E1 9507.114,E2 9507.114} C_VEL
LIN {X 0,Y 250.555,Z 815.806,A -85,B 0,C 180,E1 9504.736,E2 9504.736} C_VEL
LIN {X 0,Y 241.085,Z 830.943,A -85,B 0,C 180,E1 9501.989,E2 9501.989} C_VEL
LIN {X 0,Y 231.285,Z 844.985,A -85,B 0,C 180,E1 9498.774,E2 9498.774} C_VEL
LIN {X 0,Y 221.625,Z 857.599,A -85,B 0,C 180,E1 9495.09,E2 9495.09} C_VEL
LIN {X 0,Y 212.299,Z 868.78,A -85,B 0,C 180,E1 9490.886,E2 9490.886} C_VEL
LIN {X 0,Y 203.609,Z 878.461,A -85,B 0,C 180,E1 9486.101,E2 9486.101} C_VEL
LIN {X 0,Y 195.866,Z 886.715,A -85,B 0,C 180,E1 9480.691,E2 9480.691} C_VEL
LIN {X 0,Y 189.433,Z 893.465,A -85,B 0,C 180,E1 9474.64,E2 9474.64} C_VEL
LIN {X 0,Y 184.729,Z 898.448,A -85,B 0,C 180,E1 9468.293,E2 9468.293} C_VEL
LIN {X 0,Y 181.663,Z 901.907,A -85,B 0,C 180,E1 9461.426,E2 9461.426} C_VEL
LIN {X 0,Y 180.208,Z 903.6,A -85,B 0,C 180,E1 9454.772,E2 9454.772} C_VEL
LIN {X 0,Y 179.958,Z 903.918,A -85,B 0,C 180,E1 9448.407,E2 9448.407} C_VEL
LIN {X 0,Y 180.723,Z 903.028,A -85,B 0,C 180,E1 9442.03,E2 9442.03} C_VEL
LIN {X 0,Y 182.805,Z 900.6,A -85,B 0,C 180,E1 9435.428,E2 9435.428} C_VEL
LIN {X 0,Y 186.546,Z 896.539,A -85,B 0,C 180,E1 9428.848,E2 9428.848} C_VEL
LIN {X 0,Y 192.201,Z 890.633,A -85,B 0,C 180,E1 9422.422,E2 9422.422} C_VEL
LIN {X 0,Y 199.092,Z 883.435,A -85,B 0,C 180,E1 9416.813,E2 9416.813} C_VEL
LIN {X 0,Y 207.476,Z 874.363,A -85,B 0,C 180,E1 9411.565,E2 9411.565} C_VEL
LIN {X 0,Y 216.736,Z 863.715,A -85,B 0,C 180,E1 9406.944,E2 9406.944} C_VEL
LIN {X 0,Y 225.955,Z 852.234,A -85,B 0,C 180,E1 9403.107,E2 9403.107} C_VEL
LIN {X 0,Y 235.995,Z 838.629,A -85,B 0,C 180,E1 9399.553,E2 9399.553} C_VEL
LIN {X 0,Y 245.764,Z 823.938,A -85,B 0,C 180,E1 9396.541,E2 9396.541} C_VEL
LIN {X 0,Y 255.033,Z 808.285,A -85,B 0,C 180,E1 9393.992,E2 9393.992} C_VEL
LIN {X 0,Y 263.771,Z 791.256,A -85,B 0,C 180,E1 9391.797,E2 9391.797} C_VEL
LIN {X 0,Y 271.716,Z 773.246,A -85,B 0,C 180,E1 9389.944,E2 9389.944} C_VEL
LIN {X 0,Y 278.895,Z 753.787,A -85,B 0,C 180,E1 9388.351,E2 9388.351} C_VEL
LIN {X 0,Y 284.694,Z 734.388,A -85,B 0,C 180,E1 9387.098,E2 9387.098} C_VEL
LIN {X 0,Y 289.37,Z 714.06,A -85,B 0,C 180,E1 9386.079,E2 9386.079} C_VEL
LIN {X 0,Y 292.618,Z 693.692,A -85,B 0,C 180,E1 9385.32,E2 9385.32} C_VEL
LIN {X 0,Y 295.17,Z 667.166,A -85,B 0,C 180,E1 9384.631,E2 9384.631} C_VEL
LIN {X 0,Y 305.448,Z 551.36,A -85,B 0,C 180,E1 9382.317,E2 9382.317} C_VEL
LIN {X 0,Y 300.994,Z 543.33,A -85,B 0,C 180,E1 9379.049,E2 9379.049} C_VEL
LIN {X 0,Y 297.426,Z 537.338,A -85,B 0,C 180,E1 9375.802,E2 9375.802} C_VEL
LIN {X 0,Y 295.118,Z 533.638,A -85,B 0,C 180,E1 9373.121,E2 9373.121} C_VEL
LIN {X 0,Y 292.421,Z 529.464,A -85,B 0,C 180,E1 9368.455,E2 9368.455} C_VEL
LIN {X 0,Y 291.308,Z 528.784,A -85,B 0,C 180,E1 9363.937,E2 9363.937} C_VEL
LIN {X 0,Y 291.484,Z 529.51,A -85,B 0,C 180,E1 9360.59,E2 9360.59} C_VEL
LIN {X 0,Y 293.062,Z 533.636,A -85,B 0,C 180,E1 9355.892,E2 9355.892} C_VEL
LIN {X 0,Y 293.177,Z 533.967,A -85,B 0,C 180,E1 9355.66,E2 9355.66} C_VEL
LIN {X 0,Y 293.846,Z 536.935,A -85,B 0,C 180,E1 9354.264,E2 9354.264} C_VEL
LIN {X 0,Y 294.976,Z 545.042,A -85,B 0,C 180,E1 9351.914,E2 9351.914} C_VEL
LIN {X 0,Y 296.245,Z 551.063,A -85,B 0,C 180,E1 9350.085,E2 9350.085} C_VEL
LIN {X 0,Y 296.596,Z 552.022,A -85,B 0,C 180,E1 9349.698,E2 9349.698} C_VEL
LIN {X 0,Y 300.267,Z 560.501,A -85,B 0,C 180,E1 9346.325,E2 9346.325} C_VEL
LIN {X 0,Y 302.724,Z 566.711,A -85,B 0,C 180,E1 9344.39,E2 9344.39} C_VEL
LIN {X 0,Y 288.064,Z 717.58,A -85,B 0,C 180,E1 9341.311,E2 9341.311} C_VEL
LIN {X 0,Y 284.196,Z 739.857,A -85,B 0,C 180,E1 9340.693,E2 9340.693} C_VEL
LIN {X 0,Y 278.879,Z 761.356,A -85,B 0,C 180,E1 9339.928,E2 9339.928} C_VEL
LIN {X 0,Y 272.074,Z 782.561,A -85,B 0,C 180,E1 9338.964,E2 9338.964} C_VEL
LIN {X 0,Y 264.475,Z 802.167,A -85,B 0,C 180,E1 9337.787,E2 9337.787} C_VEL
LIN {X 0,Y 255.612,Z 821.548,A -85,B 0,C 180,E1 9336.24,E2 9336.24} C_VEL
LIN {X 0,Y 245.799,Z 840.411,A -85,B 0,C 180,E1 9334.282,E2 9334.282} C_VEL
LIN {X 0,Y 235.3,Z 858.452,A -85,B 0,C 180,E1 9331.858,E2 9331.858} C_VEL
LIN {X 0,Y 224.592,Z 875.175,A -85,B 0,C 180,E1 9328.972,E2 9328.972} C_VEL
LIN {X 0,Y 213.689,Z 890.894,A -85,B 0,C 180,E1 9325.431,E2 9325.431} C_VEL
LIN {X 0,Y 203.462,Z 904.871,A -85,B 0,C 180,E1 9321.38,E2 9321.38} C_VEL
LIN {X 0,Y 193.427,Z 918.287,A -85,B 0,C 180,E1 9316.355,E2 9316.355} C_VEL
LIN {X 0,Y 185.059,Z 929.707,A -85,B 0,C 180,E1 9310.822,E2 9310.822} C_VEL
LIN {X 0,Y 178.063,Z 939.873,A -85,B 0,C 180,E1 9304.369,E2 9304.369} C_VEL
LIN {X 0,Y 173.274,Z 948.148,A -85,B 0,C 180,E1 9297.491,E2 9297.491} C_VEL
LIN {X 0,Y 170.663,Z 954.765,A -85,B 0,C 180,E1 9290.221,E2 9290.221} C_VEL
LIN {X 0,Y 170.057,Z 959.146,A -85,B 0,C 180,E1 9283.602,E2 9283.602} C_VEL
LIN {X 0,Y 170.61,Z 961.85,A -85,B 0,C 180,E1 9277.408,E2 9277.408} C_VEL
LIN {X 0,Y 171.273,Z 962.928,A -85,B 0,C 180,E1 9272.678,E2 9272.678} C_VEL
LIN {X 0,Y 171.376,Z 963.059,A -85,B 0,C 180,E1 9268.664,E2 9268.664} C_VEL
LIN {X 0,Y 170.848,Z 962.301,A -85,B 0,C 180,E1 9264.202,E2 9264.202} C_VEL
LIN {X 0,Y 170.194,Z 960.331,A -85,B 0,C 180,E1 9258.824,E2 9258.824} C_VEL
LIN {X 0,Y 170.309,Z 956.284,A -85,B 0,C 180,E1 9251.874,E2 9251.874} C_VEL
LIN {X 0,Y 172.159,Z 950.567,A -85,B 0,C 180,E1 9244.919,E2 9244.919} C_VEL
LIN {X 0,Y 176.048,Z 943.064,A -85,B 0,C 180,E1 9238.122,E2 9238.122} C_VEL
LIN {X 0,Y 182.415,Z 933.296,A -85,B 0,C 180,E1 9231.334,E2 9231.334} C_VEL
LIN {X 0,Y 190.136,Z 922.669,A -85,B 0,C 180,E1 9225.628,E2 9225.628} C_VEL
LIN {X 0,Y 199.571,Z 910.006,A -85,B 0,C 180,E1 9220.409,E2 9220.409} C_VEL
LIN {X 0,Y 209.338,Z 896.762,A -85,B 0,C 180,E1 9216.187,E2 9216.187} C_VEL
LIN {X 0,Y 220.172,Z 881.455,A -85,B 0,C 180,E1 9212.374,E2 9212.374} C_VEL
LIN {X 0,Y 230.662,Z 865.725,A -85,B 0,C 180,E1 9209.328,E2 9209.328} C_VEL
LIN {X 0,Y 241.202,Z 848.304,A -85,B 0,C 180,E1 9206.721,E2 9206.721} C_VEL
LIN {X 0,Y 251.229,Z 829.958,A -85,B 0,C 180,E1 9204.592,E2 9204.592} C_VEL
LIN {X 0,Y 260.431,Z 810.952,A -85,B 0,C 180,E1 9202.881,E2 9202.881} C_VEL
LIN {X 0,Y 268.686,Z 791.318,A -85,B 0,C 180,E1 9201.531,E2 9201.531} C_VEL
LIN {X 0,Y 275.876,Z 770.797,A -85,B 0,C 180,E1 9200.483,E2 9200.483} C_VEL
LIN {X 0,Y 281.939,Z 749.05,A -85,B 0,C 180,E1 9199.628,E2 9199.628} C_VEL
LIN {X 0,Y 286.471,Z 726.739,A -85,B 0,C 180,E1 9198.942,E2 9198.942} C_VEL
LIN {X 0,Y 289.392,Z 704.19,A -85,B 0,C 180,E1 9198.407,E2 9198.407} C_VEL
LIN {X 0,Y 302.524,Z 566.215,A -85,B 0,C 180,E1 9195.582,E2 9195.582} C_VEL
LIN {X 0,Y 298.602,Z 556.926,A -85,B 0,C 180,E1 9192.423,E2 9192.423} C_VEL
LIN {X 0,Y 295.662,Z 550.323,A -85,B 0,C 180,E1 9189.538,E2 9189.538} C_VEL
LIN {X 0,Y 293.427,Z 545.231,A -85,B 0,C 180,E1 9186.751,E2 9186.751} C_VEL
LIN {X 0,Y 291.346,Z 540.391,A -85,B 0,C 180,E1 9183.076,E2 9183.076} C_VEL
LIN {X 0,Y 290.197,Z 536.955,A -85,B 0,C 180,E1 9178.815,E2 9178.815} C_VEL
LIN {X 0,Y 290.469,Z 536.63,A -85,B 0,C 180,E1 9173.676,E2 9173.676} C_VEL
LIN {X 0,Y 291.542,Z 537.705,A -85,B 0,C 180,E1 9170.724,E2 9170.724} C_VEL
LIN {X 0,Y 294.322,Z 542.228,A -85,B 0,C 180,E1 9166.243,E2 9166.243} C_VEL
LIN {X 0,Y 296.922,Z 546.678,A -85,B 0,C 180,E1 9163.367,E2 9163.367} C_VEL
LIN {X 0,Y 300.202,Z 552.388,A -85,B 0,C 180,E1 9160.487,E2 9160.487} C_VEL
LIN {X 0,Y 302.286,Z 556.677,A -85,B 0,C 180,E1 9158.869,E2 9158.869} C_VEL
LIN {X 0,Y 290.683,Z 683.185,A -85,B 0,C 180,E1 9156.353,E2 9156.353} C_VEL
LIN {X 0,Y 288.006,Z 704.154,A -85,B 0,C 180,E1 9155.703,E2 9155.703} C_VEL
LIN {X 0,Y 283.791,Z 725.352,A -85,B 0,C 180,E1 9154.796,E2 9154.796} C_VEL
LIN {X 0,Y 278.709,Z 744.156,A -85,B 0,C 180,E1 9153.736,E2 9153.736} C_VEL
LIN {X 0,Y 272.036,Z 763.872,A -85,B 0,C 180,E1 9152.336,E2 9152.336} C_VEL
LIN {X 0,Y 264.718,Z 781.76,A -85,B 0,C 180,E1 9150.739,E2 9150.739} C_VEL
LIN {X 0,Y 256.1,Z 799.549,A -85,B 0,C 180,E1 9148.75,E2 9148.75} C_VEL
LIN {X 0,Y 247.022,Z 815.641,A -85,B 0,C 180,E1 9146.482,E2 9146.482} C_VEL
LIN {X 0,Y 236.962,Z 831.374,A -85,B 0,C 180,E1 9143.69,E2 9143.69} C_VEL
LIN {X 0,Y 226.77,Z 845.559,A -85,B 0,C 180,E1 9140.489,E2 9140.489} C_VEL
LIN {X 0,Y 216.679,Z 858.3,A -85,B 0,C 180,E1 9136.802,E2 9136.802} C_VEL
LIN {X 0,Y 206.881,Z 869.544,A -85,B 0,C 180,E1 9132.574,E2 9132.574} C_VEL
LIN {X 0,Y 197.698,Z 879.334,A -85,B 0,C 180,E1 9127.725,E2 9127.725} C_VEL
LIN {X 0,Y 189.455,Z 887.69,A -85,B 0,C 180,E1 9122.206,E2 9122.206} C_VEL
LIN {X 0,Y 182.532,Z 894.533,A -85,B 0,C 180,E1 9115.986,E2 9115.986} C_VEL
LIN {X 0,Y 177.418,Z 899.604,A -85,B 0,C 180,E1 9109.417,E2 9109.417} C_VEL
LIN {X 0,Y 174.024,Z 903.108,A -85,B 0,C 180,E1 9102.271,E2 9102.271} C_VEL
LIN {X 0,Y 172.383,Z 904.87,A -85,B 0,C 180,E1 9095.323,E2 9095.323} C_VEL
LIN {X 0,Y 172.071,Z 905.246,A -85,B 0,C 180,E1 9088.334,E2 9088.334} C_VEL
LIN {X 0,Y 172.895,Z 904.364,A -85,B 0,C 180,E1 9081.687,E2 9081.687} C_VEL
LIN {X 0,Y 175.174,Z 901.907,A -85,B 0,C 180,E1 9074.716,E2 9074.716} C_VEL
LIN {X 0,Y 179.091,Z 897.948,A -85,B 0,C 180,E1 9068.035,E2 9068.035} C_VEL
LIN {X 0,Y 185.199,Z 891.971,A -85,B 0,C 180,E1 9061.284,E2 9061.284} C_VEL
LIN {X 0,Y 192.496,Z 884.776,A -85,B 0,C 180,E1 9055.519,E2 9055.519} C_VEL
LIN {X 0,Y 201.32,Z 875.711,A -85,B 0,C 180,E1 9050.161,E2 9050.161} C_VEL
LIN {X 0,Y 211.015,Z 865.063,A -85,B 0,C 180,E1 9045.475,E2 9045.475} C_VEL
LIN {X 0,Y 220.621,Z 853.594,A -85,B 0,C 180,E1 9041.607,E2 9041.607} C_VEL
LIN {X 0,Y 231.044,Z 840.005,A -85,B 0,C 180,E1 9038.043,E2 9038.043} C_VEL
LIN {X 0,Y 241.151,Z 825.34,A -85,B 0,C 180,E1 9035.035,E2 9035.035} C_VEL
LIN {X 0,Y 250.79,Z 809.582,A -85,B 0,C 180,E1 9032.481,E2 9032.481} C_VEL
LIN {X 0,Y 259.542,Z 793.053,A -85,B 0,C 180,E1 9030.361,E2 9030.361} C_VEL
LIN {X 0,Y 267.516,Z 775.647,A -85,B 0,C 180,E1 9028.568,E2 9028.568} C_VEL
LIN {X 0,Y 274.745,Z 756.949,A -85,B 0,C 180,E1 9027.022,E2 9027.022} C_VEL
LIN {X 0,Y 280.964,Z 737.181,A -85,B 0,C 180,E1 9025.732,E2 9025.732} C_VEL
LIN {X 0,Y 285.849,Z 716.764,A -85,B 0,C 180,E1 9024.703,E2 9024.703} C_VEL
LIN {X 0,Y 289.337,Z 696.331,A -85,B 0,C 180,E1 9023.928,E2 9023.928} C_VEL
LIN {X 0,Y 292.013,Z 670.498,A -85,B 0,C 180,E1 9023.243,E2 9023.243} C_VEL
LIN {X 0,Y 302.476,Z 556.549,A -85,B 0,C 180,E1 9021.018,E2 9021.018} C_VEL
LIN {X 0,Y 298.541,Z 549.172,A -85,B 0,C 180,E1 9017.846,E2 9017.846} C_VEL
LIN {X 0,Y 295.647,Z 544.392,A -85,B 0,C 180,E1 9014.994,E2 9014.994} C_VEL
LIN {X 0,Y 293.861,Z 541.364,A -85,B 0,C 180,E1 9012.778,E2 9012.778} C_VEL
LIN {X 0,Y 291.379,Z 537.361,A -85,B 0,C 180,E1 9008.287,E2 9008.287} C_VEL
LIN {X 0,Y 290.322,Z 536.73,A -85,B 0,C 180,E1 9003.752,E2 9003.752} C_VEL
LIN {X 0,Y 290.474,Z 537.39,A -85,B 0,C 180,E1 9000.789,E2 9000.789} C_VEL
LIN {X 0,Y 291.907,Z 541.448,A -85,B 0,C 180,E1 8996.171,E2 8996.171} C_VEL
LIN {X 0,Y 293.904,Z 546.076,A -85,B 0,C 180,E1 8992.868,E2 8992.868} C_VEL
LIN {X 0,Y 296.453,Z 551.67,A -85,B 0,C 180,E1 8989.85,E2 8989.85} C_VEL
LIN {X 0,Y 296.596,Z 552.022,A -85,B 0,C 180,E1 8989.698,E2 8989.698} C_VEL
LIN {X 0,Y 297.255,Z 555.004,A -85,B 0,C 180,E1 8988.885,E2 8988.885} C_VEL
LIN {X 0,Y 298.351,Z 566.763,A -85,B 0,C 180,E1 8987.036,E2 8987.036} C_VEL
LIN {X 0,Y 298.937,Z 568.999,A -85,B 0,C 180,E1 8986.464,E2 8986.464} C_VEL
LIN {X 0,Y 299.775,Z 571.357,A -85,B 0,C 180,E1 8985.747,E2 8985.747} C_VEL
LIN {X 0,Y 285.309,Z 716.521,A -85,B 0,C 180,E1 8982.83,E2 8982.83} C_VEL
LIN {X 0,Y 281.394,Z 738.655,A -85,B 0,C 180,E1 8982.231,E2 8982.231} C_VEL
LIN {X 0,Y 275.971,Z 760.219,A -85,B 0,C 180,E1 8981.487,E2 8981.487} C_VEL
LIN {X 0,Y 269.252,Z 780.854,A -85,B 0,C 180,E1 8980.585,E2 8980.585} C_VEL
LIN {X 0,Y 261.564,Z 800.326,A -85,B 0,C 180,E1 8979.465,E2 8979.465} C_VEL
LIN {X 0,Y 252.81,Z 819.137,A -85,B 0,C 180,E1 8978.027,E2 8978.027} C_VEL
LIN {X 0,Y 242.483,Z 838.602,A -85,B 0,C 180,E1 8976.081,E2 8976.081} C_VEL
LIN {X 0,Y 231.844,Z 856.421,A -85,B 0,C 180,E1 8973.76,E2 8973.76} C_VEL
LIN {X 0,Y 220.757,Z 873.183,A -85,B 0,C 180,E1 8970.935,E2 8970.935} C_VEL
LIN {X 0,Y 209.692,Z 888.525,A -85,B 0,C 180,E1 8967.555,E2 8967.555} C_VEL
LIN {X 0,Y 198.301,Z 903.424,A -85,B 0,C 180,E1 8963.287,E2 8963.287} C_VEL
LIN {X 0,Y 187.696,Z 916.852,A -85,B 0,C 180,E1 8958.221,E2 8958.221} C_VEL
LIN {X 0,Y 178.743,Z 928.276,A -85,B 0,C 180,E1 8952.594,E2 8952.594} C_VEL
LIN {X 0,Y 171.309,Z 938.232,A -85,B 0,C 180,E1 8946.118,E2 8946.118} C_VEL
LIN {X 0,Y 166.082,Z 946.373,A -85,B 0,C 180,E1 8939.184,E2 8939.184} C_VEL
LIN {X 0,Y 163.076,Z 952.846,A -85,B 0,C 180,E1 8931.962,E2 8931.962} C_VEL
LIN {X 0,Y 162.129,Z 957.357,A -85,B 0,C 180,E1 8925.011,E2 8925.011} C_VEL
LIN {X 0,Y 162.595,Z 960.405,A -85,B 0,C 180,E1 8918.095,E2 8918.095} C_VEL
LIN {X 0,Y 163.358,Z 961.594,A -85,B 0,C 180,E1 8912.808,E2 8912.808} C_VEL
LIN {X 0,Y 163.478,Z 961.729,A -85,B 0,C 180,E1 8908.6,E2 8908.6} C_VEL
LIN {X 0,Y 162.893,Z 960.953,A -85,B 0,C 180,E1 8903.913,E2 8903.913} C_VEL
LIN {X 0,Y 162.225,Z 958.962,A -85,B 0,C 180,E1 8898.267,E2 8898.267} C_VEL
LIN {X 0,Y 162.472,Z 954.891,A -85,B 0,C 180,E1 8890.967,E2 8890.967} C_VEL
LIN {X 0,Y 164.785,Z 948.845,A -85,B 0,C 180,E1 8883.324,E2 8883.324} C_VEL
LIN {X 0,Y 169.508,Z 940.812,A -85,B 0,C 180,E1 8875.924,E2 8875.924} C_VEL
LIN {X 0,Y 176.286,Z 931.341,A -85,B 0,C 180,E1 8869.295,E2 8869.295} C_VEL
LIN {X 0,Y 185.159,Z 919.95,A -85,B 0,C 180,E1 8863.205,E2 8863.205} C_VEL
LIN {X 0,Y 195.357,Z 907.139,A -85,B 0,C 180,E1 8857.993,E2 8857.993} C_VEL
LIN {X 0,Y 206.403,Z 892.806,A -85,B 0,C 180,E1 8853.581,E2 8853.581} C_VEL
LIN {X 0,Y 217.539,Z 877.512,A -85,B 0,C 180,E1 8849.97,E2 8849.97} C_VEL
LIN {X 0,Y 229.186,Z 860.322,A -85,B 0,C 180,E1 8846.867,E2 8846.867} C_VEL
LIN {X 0,Y 239.799,Z 843.085,A -85,B 0,C 180,E1 8844.466,E2 8844.466} C_VEL
LIN {X 0,Y 249.939,Z 824.597,A -85,B 0,C 180,E1 8842.484,E2 8842.484} C_VEL
LIN {X 0,Y 259.025,Z 805.632,A -85,B 0,C 180,E1 8840.928,E2 8840.928} C_VEL
LIN {X 0,Y 267.516,Z 785.046,A -85,B 0,C 180,E1 8839.651,E2 8839.651} C_VEL
LIN {X 0,Y 274.439,Z 764.925,A -85,B 0,C 180,E1 8838.712,E2 8838.712} C_VEL
LIN {X 0,Y 280.357,Z 742.712,A -85,B 0,C 180,E1 8837.907,E2 8837.907} C_VEL
LIN {X 0,Y 284.473,Z 720.728,A -85,B 0,C 180,E1 8837.29,E2 8837.29} C_VEL
LIN {X 0,Y 287.951,Z 689.914,A -85,B 0,C 180,E1 8836.625,E2 8836.625} C_VEL
LIN {X 0,Y 299.599,Z 570.999,A -85,B 0,C 180,E1 8834.248,E2 8834.248} C_VEL
LIN {X 0,Y 296.456,Z 563.225,A -85,B 0,C 180,E1 8831.477,E2 8831.477} C_VEL
LIN {X 0,Y 293.784,Z 556.907,A -85,B 0,C 180,E1 8828.612,E2 8828.612} C_VEL
LIN {X 0,Y 291.764,Z 551.989,A -85,B 0,C 180,E1 8825.802,E2 8825.802} C_VEL
LIN {X 0,Y 290.208,Z 548.167,A -85,B 0,C 180,E1 8822.764,E2 8822.764} C_VEL
LIN {X 0,Y 289.188,Z 544.852,A -85,B 0,C 180,E1 8818.613,E2 8818.613} C_VEL
LIN {X 0,Y 289.498,Z 544.581,A -85,B 0,C 180,E1 8813.654,E2 8813.654} C_VEL
LIN {X 0,Y 290.479,Z 545.61,A -85,B 0,C 180,E1 8810.889,E2 8810.889} C_VEL
LIN {X 0,Y 293.122,Z 550.087,A -85,B 0,C 180,E1 8806.487,E2 8806.487} C_VEL
LIN {X 0,Y 295.566,Z 554.418,A -85,B 0,C 180,E1 8803.693,E2 8803.693} C_VEL
LIN {X 0,Y 298.632,Z 560.007,A -85,B 0,C 180,E1 8800.896,E2 8800.896} C_VEL
LIN {X 0,Y 299.411,Z 561.916,A -85,B 0,C 180,E1 8800.227,E2 8800.227} C_VEL
LIN {X 0,Y 287.898,Z 683.82,A -85,B 0,C 180,E1 8797.833,E2 8797.833} C_VEL
LIN {X 0,Y 285.142,Z 704.926,A -85,B 0,C 180,E1 8797.188,E2 8797.188} C_VEL
LIN {X 0,Y 280.814,Z 726.143,A -85,B 0,C 180,E1 8796.295,E2 8796.295} C_VEL
LIN {X 0,Y 275.334,Z 745.887,A -85,B 0,C 180,E1 8795.197,E2 8795.197} C_VEL
LIN {X 0,Y 268.484,Z 765.463,A -85,B 0,C 180,E1 8793.818,E2 8793.818} C_VEL
LIN {X 0,Y 260.967,Z 783.262,A -85,B 0,C 180,E1 8792.244,E2 8792.244} C_VEL
LIN {X 0,Y 252.11,Z 801.019,A -85,B 0,C 180,E1 8790.278,E2 8790.278} C_VEL
LIN {X 0,Y 242.431,Z 817.612,A -85,B 0,C 180,E1 8787.948,E2 8787.948} C_VEL
LIN {X 0,Y 232.376,Z 832.766,A -85,B 0,C 180,E1 8785.258,E2 8785.258} C_VEL
LIN {X 0,Y 221.825,Z 846.931,A -85,B 0,C 180,E1 8782.065,E2 8782.065} C_VEL
LIN {X 0,Y 211.339,Z 859.656,A -85,B 0,C 180,E1 8778.367,E2 8778.367} C_VEL
LIN {X 0,Y 201.116,Z 870.899,A -85,B 0,C 180,E1 8774.101,E2 8774.101} C_VEL
LIN {X 0,Y 191.483,Z 880.68,A -85,B 0,C 180,E1 8769.178,E2 8769.178} C_VEL
LIN {X 0,Y 182.787,Z 889.03,A -85,B 0,C 180,E1 8763.532,E2 8763.532} C_VEL
LIN {X 0,Y 175.431,Z 895.872,A -85,B 0,C 180,E1 8757.122,E2 8757.122} C_VEL
LIN {X 0,Y 169.957,Z 900.939,A -85,B 0,C 180,E1 8750.306,E2 8750.306} C_VEL
LIN {X 0,Y 166.299,Z 904.442,A -85,B 0,C 180,E1 8742.851,E2 8742.851} C_VEL
LIN {X 0,Y 164.524,Z 906.2,A -85,B 0,C 180,E1 8735.578,E2 8735.578} C_VEL
LIN {X 0,Y 164.184,Z 906.574,A -85,B 0,C 180,E1 8728.254,E2 8728.254} C_VEL
LIN {X 0,Y 165.079,Z 905.695,A -85,B 0,C 180,E1 8721.29,E2 8721.29} C_VEL
LIN {X 0,Y 167.512,Z 903.266,A -85,B 0,C 180,E1 8714.064,E2 8714.064} C_VEL
LIN {X 0,Y 171.755,Z 899.284,A -85,B 0,C 180,E1 8707.045,E2 8707.045} C_VEL
LIN {X 0,Y 178.273,Z 893.31,A -85,B 0,C 180,E1 8700.057,E2 8700.057} C_VEL
LIN {X 0,Y 186.005,Z 886.119,A -85,B 0,C 180,E1 8694.135,E2 8694.135} C_VEL
LIN {X 0,Y 195.293,Z 877.059,A -85,B 0,C 180,E1 8688.669,E2 8688.669} C_VEL
LIN {X 0,Y 205.44,Z 866.411,A -85,B 0,C 180,E1 8683.925,E2 8683.925} C_VEL
LIN {X 0,Y 215.448,Z 854.953,A -85,B 0,C 180,E1 8680.033,E2 8680.033} C_VEL
LIN {X 0,Y 226.261,Z 841.38,A -85,B 0,C 180,E1 8676.467,E2 8676.467} C_VEL
LIN {X 0,Y 236.711,Z 826.741,A -85,B 0,C 180,E1 8673.471,E2 8673.471} C_VEL
LIN {X 0,Y 246.572,Z 811.13,A -85,B 0,C 180,E1 8670.956,E2 8670.956} C_VEL
LIN {X 0,Y 255.657,Z 794.515,A -85,B 0,C 180,E1 8668.839,E2 8668.839} C_VEL
LIN {X 0,Y 264.069,Z 776.674,A -85,B 0,C 180,E1 8667.024,E2 8667.024} C_VEL
LIN {X 0,Y 271.419,Z 758.163,A -85,B 0,C 180,E1 8665.517,E2 8665.517} C_VEL
LIN {X 0,Y 277.768,Z 738.55,A -85,B 0,C 180,E1 8664.254,E2 8664.254} C_VEL
LIN {X 0,Y 282.788,Z 718.191,A -85,B 0,C 180,E1 8663.238,E2 8663.238} C_VEL
LIN {X 0,Y 286.424,Z 697.651,A -85,B 0,C 180,E1 8662.464,E2 8662.464} C_VEL
LIN {X 0,Y 289.2,Z 671.931,A -85,B 0,C 180,E1 8661.784,E2 8661.784} C_VEL
LIN {X 0,Y 299.603,Z 561.734,A -85,B 0,C 180,E1 8659.653,E2 8659.653} C_VEL
LIN {X 0,Y 296.326,Z 555.598,A -85,B 0,C 180,E1 8656.768,E2 8656.768} C_VEL
LIN {X 0,Y 294.172,Z 551.829,A -85,B 0,C 180,E1 8654.467,E2 8654.467} C_VEL
LIN {X 0,Y 292.615,Z 549.089,A -85,B 0,C 180,E1 8652.432,E2 8652.432} C_VEL
LIN {X 0,Y 290.34,Z 545.259,A -85,B 0,C 180,E1 8648.117,E2 8648.117} C_VEL
LIN {X 0,Y 289.34,Z 544.677,A -85,B 0,C 180,E1 8643.567,E2 8643.567} C_VEL
LIN {X 0,Y 289.467,Z 545.269,A -85,B 0,C 180,E1 8640.99,E2 8640.99} C_VEL
LIN {X 0,Y 290.719,Z 549.122,A -85,B 0,C 180,E1 8636.55,E2 8636.55} C_VEL
LIN {X 0,Y 292.608,Z 553.76,A -85,B 0,C 180,E1 8633.23,E2 8633.23} C_VEL
LIN {X 0,Y 295.044,Z 559.446,A -85,B 0,C 180,E1 8630.196,E2 8630.196} C_VEL
LIN {X 0,Y 298.4,Z 567.627,A -85,B 0,C 180,E1 8626.929,E2 8626.929} C_VEL
LIN {X 0,Y 298.937,Z 568.999,A -85,B 0,C 180,E1 8626.464,E2 8626.464} C_VEL
LIN {X 0,Y 299.167,Z 570.954,A -85,B 0,C 180,E1 8626.157,E2 8626.157} C_VEL
LIN {X 0,Y 298.916,Z 574.289,A -85,B 0,C 180,E1 8626.041,E2 8626.041} C_VEL
LIN {X 0,Y 298.009,Z 579.295,A -85,B 0,C 180,E1 8626.198,E2 8626.198} C_VEL
LIN {X 0,Y 295.798,Z 589.217,A -85,B 0,C 180,E1 8626.788,E2 8626.788} C_VEL
LIN {X 0,Y 295.312,Z 592.655,A -85,B 0,C 180,E1 8626.812,E2 8626.812} C_VEL
LIN {X 0,Y 282.734,Z 715.671,A -85,B 0,C 180,E1 8624.372,E2 8624.372} C_VEL
LIN {X 0,Y 278.684,Z 738.016,A -85,B 0,C 180,E1 8623.782,E2 8623.782} C_VEL
LIN {X 0,Y 273.272,Z 759.083,A -85,B 0,C 180,E1 8623.078,E2 8623.078} C_VEL
LIN {X 0,Y 266.212,Z 780.303,A -85,B 0,C 180,E1 8622.182,E2 8622.182} C_VEL
LIN {X 0,Y 258.373,Z 799.703,A -85,B 0,C 180,E1 8621.101,E2 8621.101} C_VEL
LIN {X 0,Y 249.004,Z 819.248,A -85,B 0,C 180,E1 8619.639,E2 8619.639} C_VEL
LIN {X 0,Y 238.666,Z 838.073,A -85,B 0,C 180,E1 8617.785,E2 8617.785} C_VEL
LIN {X 0,Y 227.501,Z 856.109,A -85,B 0,C 180,E1 8615.461,E2 8615.461} C_VEL
LIN {X 0,Y 216.076,Z 872.755,A -85,B 0,C 180,E1 8612.67,E2 8612.67} C_VEL
LIN {X 0,Y 204.613,Z 887.978,A -85,B 0,C 180,E1 8609.313,E2 8609.313} C_VEL
LIN {X 0,Y 193.375,Z 901.978,A -85,B 0,C 180,E1 8605.291,E2 8605.291} C_VEL
LIN {X 0,Y 182.727,Z 914.78,A -85,B 0,C 180,E1 8600.486,E2 8600.486} C_VEL
LIN {X 0,Y 172.606,Z 926.843,A -85,B 0,C 180,E1 8594.497,E2 8594.497} C_VEL
LIN {X 0,Y 164.524,Z 936.858,A -85,B 0,C 180,E1 8587.812,E2 8587.812} C_VEL
LIN {X 0,Y 158.579,Z 945.32,A -85,B 0,C 180,E1 8580.29,E2 8580.29} C_VEL
LIN {X 0,Y 155.178,Z 951.968,A -85,B 0,C 180,E1 8572.342,E2 8572.342} C_VEL
LIN {X 0,Y 154.183,Z 956.442,A -85,B 0,C 180,E1 8564.932,E2 8564.932} C_VEL
LIN {X 0,Y 154.716,Z 959.243,A -85,B 0,C 180,E1 8557.8,E2 8557.8} C_VEL
LIN {X 0,Y 155.483,Z 960.298,A -85,B 0,C 180,E1 8552.581,E2 8552.581} C_VEL
LIN {X 0,Y 155.579,Z 960.398,A -85,B 0,C 180,E1 8548.528,E2 8548.528} C_VEL
LIN {X 0,Y 154.932,Z 959.613,A -85,B 0,C 180,E1 8543.632,E2 8543.632} C_VEL
LIN {X 0,Y 154.257,Z 957.59,A -85,B 0,C 180,E1 8537.652,E2 8537.652} C_VEL
LIN {X 0,Y 154.67,Z 953.495,A -85,B 0,C 180,E1 8529.967,E2 8529.967} C_VEL
LIN {X 0,Y 157.344,Z 947.433,A -85,B 0,C 180,E1 8521.955,E2 8521.955} C_VEL
LIN {X 0,Y 162.593,Z 939.388,A -85,B 0,C 180,E1 8514.259,E2 8514.259} C_VEL
LIN {X 0,Y 170.222,Z 929.595,A -85,B 0,C 180,E1 8507.241,E2 8507.241} C_VEL
LIN {X 0,Y 180.003,Z 917.87,A -85,B 0,C 180,E1 8500.945,E2 8500.945} C_VEL
LIN {X 0,Y 190.276,Z 905.686,A -85,B 0,C 180,E1 8495.989,E2 8495.989} C_VEL
LIN {X 0,Y 201.868,Z 891.353,A -85,B 0,C 180,E1 8491.59,E2 8491.59} C_VEL
LIN {X 0,Y 213.531,Z 875.975,A -85,B 0,C 180,E1 8488.009,E2 8488.009} C_VEL
LIN {X 0,Y 225.425,Z 859.014,A -85,B 0,C 180,E1 8485.007,E2 8485.007} C_VEL
LIN {X 0,Y 236.224,Z 842.01,A -85,B 0,C 180,E1 8482.689,E2 8482.689} C_VEL
LIN {X 0,Y 246.485,Z 823.814,A -85,B 0,C 180,E1 8480.787,E2 8480.787} C_VEL
LIN {X 0,Y 255.782,Z 804.946,A -85,B 0,C 180,E1 8479.279,E2 8479.279} C_VEL
LIN {X 0,Y 264.445,Z 784.483,A -85,B 0,C 180,E1 8478.047,E2 8478.047} C_VEL
LIN {X 0,Y 271.622,Z 764.089,A -85,B 0,C 180,E1 8477.126,E2 8477.126} C_VEL
LIN {X 0,Y 277.628,Z 741.978,A -85,B 0,C 180,E1 8476.35,E2 8476.35} C_VEL
LIN {X 0,Y 281.826,Z 720.134,A -85,B 0,C 180,E1 8475.751,E2 8475.751} C_VEL
LIN {X 0,Y 285.357,Z 689.924,A -85,B 0,C 180,E1 8475.109,E2 8475.109} C_VEL
LIN {X 0,Y 296.789,Z 575.713,A -85,B 0,C 180,E1 8472.847,E2 8472.847} C_VEL
LIN {X 0,Y 293.913,Z 568.217,A -85,B 0,C 180,E1 8469.991,E2 8469.991} C_VEL
LIN {X 0,Y 291.234,Z 561.578,A -85,B 0,C 180,E1 8466.604,E2 8466.604} C_VEL
LIN {X 0,Y 289.659,Z 557.659,A -85,B 0,C 180,E1 8463.859,E2 8463.859} C_VEL
LIN {X 0,Y 288.973,Z 555.732,A -85,B 0,C 180,E1 8462.181,E2 8462.181} C_VEL
LIN {X 0,Y 288.179,Z 552.749,A -85,B 0,C 180,E1 8458.409,E2 8458.409} C_VEL
LIN {X 0,Y 288.528,Z 552.533,A -85,B 0,C 180,E1 8453.633,E2 8453.633} C_VEL
LIN {X 0,Y 289.422,Z 553.514,A -85,B 0,C 180,E1 8451.056,E2 8451.056} C_VEL
LIN {X 0,Y 291.857,Z 557.797,A -85,B 0,C 180,E1 8446.831,E2 8446.831} C_VEL
LIN {X 0,Y 294.129,Z 561.98,A -85,B 0,C 180,E1 8444.118,E2 8444.118} C_VEL
LIN {X 0,Y 296.723,Z 566.867,A -85,B 0,C 180,E1 8441.619,E2 8441.619} C_VEL
LIN {X 0,Y 285.286,Z 684.671,A -85,B 0,C 180,E1 8439.336,E2 8439.336} C_VEL
LIN {X 0,Y 282.448,Z 705.825,A -85,B 0,C 180,E1 8438.698,E2 8438.698} C_VEL
LIN {X 0,Y 278.008,Z 727.042,A -85,B 0,C 180,E1 8437.821,E2 8437.821} C_VEL
LIN {X 0,Y 272.531,Z 746.369,A -85,B 0,C 180,E1 8436.77,E2 8436.77} C_VEL
LIN {X 0,Y 265.505,Z 766.081,A -85,B 0,C 180,E1 8435.416,E2 8435.416} C_VEL
LIN {X 0,Y 257.787,Z 783.982,A -85,B 0,C 180,E1 8433.87,E2 8433.87} C_VEL
LIN {X 0,Y 248.666,Z 801.807,A -85,B 0,C 180,E1 8431.936,E2 8431.936} C_VEL
LIN {X 0,Y 238.684,Z 818.49,A -85,B 0,C 180,E1 8429.637,E2 8429.637} C_VEL
LIN {X 0,Y 228.673,Z 833.193,A -85,B 0,C 180,E1 8427.078,E2 8427.078} C_VEL
LIN {X 0,Y 218.392,Z 846.703,A -85,B 0,C 180,E1 8424.121,E2 8424.121} C_VEL
LIN {X 0,Y 207.404,Z 859.637,A -85,B 0,C 180,E1 8420.465,E2 8420.465} C_VEL
LIN {X 0,Y 196.633,Z 871.068,A -85,B 0,C 180,E1 8416.217,E2 8416.217} C_VEL
LIN {X 0,Y 186.4,Z 881.078,A -85,B 0,C 180,E1 8411.276,E2 8411.276} C_VEL
LIN {X 0,Y 177.073,Z 889.633,A -85,B 0,C 180,E1 8405.557,E2 8405.557} C_VEL
LIN {X 0,Y 169.4,Z 896.399,A -85,B 0,C 180,E1 8399.329,E2 8399.329} C_VEL
LIN {X 0,Y 163.255,Z 901.644,A -85,B 0,C 180,E1 8392.313,E2 8392.313} C_VEL
LIN {X 0,Y 159.145,Z 905.219,A -85,B 0,C 180,E1 8384.924,E2 8384.924} C_VEL
LIN {X 0,Y 156.841,Z 907.355,A -85,B 0,C 180,E1 8376.955,E2 8376.955} C_VEL
LIN {X 0,Y 156.274,Z 907.983,A -85,B 0,C 180,E1 8369.632,E2 8369.632} C_VEL
LIN {X 0,Y 156.96,Z 907.271,A -85,B 0,C 180,E1 8362.312,E2 8362.312} C_VEL
LIN {X 0,Y 159.266,Z 905.149,A -85,B 0,C 180,E1 8354.712,E2 8354.712} C_VEL
LIN {X 0,Y 163.451,Z 901.522,A -85,B 0,C 180,E1 8347.334,E2 8347.334} C_VEL
LIN {X 0,Y 169.677,Z 896.239,A -85,B 0,C 180,E1 8340.333,E2 8340.333} C_VEL
LIN {X 0,Y 177.86,Z 889.059,A -85,B 0,C 180,E1 8333.827,E2 8333.827} C_VEL
LIN {X 0,Y 187.327,Z 880.332,A -85,B 0,C 180,E1 8328.153,E2 8328.153} C_VEL
LIN {X 0,Y 197.683,Z 870.131,A -85,B 0,C 180,E1 8323.258,E2 8323.258} C_VEL
LIN {X 0,Y 208.548,Z 858.487,A -85,B 0,C 180,E1 8319.047,E2 8319.047} C_VEL
LIN {X 0,Y 219.632,Z 845.389,A -85,B 0,C 180,E1 8315.431,E2 8315.431} C_VEL
LIN {X 0,Y 231.041,Z 830.204,A -85,B 0,C 180,E1 8312.223,E2 8312.223} C_VEL
LIN {X 0,Y 241.135,Z 814.877,A -85,B 0,C 180,E1 8309.702,E2 8309.702} C_VEL
LIN {X 0,Y 250.783,Z 798.169,A -85,B 0,C 180,E1 8307.524,E2 8307.524} C_VEL
LIN {X 0,Y 259.603,Z 780.448,A -85,B 0,C 180,E1 8305.688,E2 8305.688} C_VEL
LIN {X 0,Y 267.359,Z 761.953,A -85,B 0,C 180,E1 8304.158,E2 8304.158} C_VEL
LIN {X 0,Y 274.003,Z 742.306,A -85,B 0,C 180,E1 8302.881,E2 8302.881} C_VEL
LIN {X 0,Y 279.359,Z 722.006,A -85,B 0,C 180,E1 8301.846,E2 8301.846} C_VEL
LIN {X 0,Y 283.533,Z 700.081,A -85,B 0,C 180,E1 8301.006,E2 8301.006} C_VEL
LIN {X 0,Y 286.187,Z 677.629,A -85,B 0,C 180,E1 8300.392,E2 8300.392} C_VEL
LIN {X 0,Y 296.886,Z 566.954,A -85,B 0,C 180,E1 8298.253,E2 8298.253} C_VEL
LIN {X 0,Y 293.545,Z 560.57,A -85,B 0,C 180,E1 8294.902,E2 8294.902} C_VEL
LIN {X 0,Y 291.344,Z 556.774,A -85,B 0,C 180,E1 8292.041,E2 8292.041} C_VEL
LIN {X 0,Y 289.303,Z 553.159,A -85,B 0,C 180,E1 8287.947,E2 8287.947} C_VEL
LIN {X 0,Y 288.367,Z 552.617,A -85,B 0,C 180,E1 8283.579,E2 8283.579} C_VEL
LIN {X 0,Y 288.464,Z 553.148,A -85,B 0,C 180,E1 8281.192,E2 8281.192} C_VEL
LIN {X 0,Y 289.592,Z 556.934,A -85,B 0,C 180,E1 8276.834,E2 8276.834} C_VEL
LIN {X 0,Y 291.321,Z 561.443,A -85,B 0,C 180,E1 8273.596,E2 8273.596} C_VEL
LIN {X 0,Y 293.767,Z 567.543,A -85,B 0,C 180,E1 8270.4,E2 8270.4} C_VEL
LIN {X 0,Y 296.668,Z 575.03,A -85,B 0,C 180,E1 8267.445,E2 8267.445} C_VEL
LIN {X 0,Y 296.98,Z 576.238,A -85,B 0,C 180,E1 8267.127,E2 8267.127} C_VEL
LIN {X 0,Y 295.312,Z 592.655,A -85,B 0,C 180,E1 8266.812,E2 8266.812} C_VEL
LIN {X 0,Y 294.246,Z 600.346,A -85,B 0,C 180,E1 8266.855,E2 8266.855} C_VEL
LIN {X 0,Y 290.433,Z 620.858,A -85,B 0,C 180,E1 8267.645,E2 8267.645} C_VEL
LIN {X 0,Y 289.556,Z 627.457,A -85,B 0,C 180,E1 8267.661,E2 8267.661} C_VEL
LIN {X 0,Y 280.338,Z 715.003,A -85,B 0,C 180,E1 8265.938,E2 8265.938} C_VEL
LIN {X 0,Y 276.155,Z 737.506,A -85,B 0,C 180,E1 8265.36,E2 8265.36} C_VEL
LIN {X 0,Y 270.564,Z 758.702,A -85,B 0,C 180,E1 8264.672,E2 8264.672} C_VEL
LIN {X 0,Y 263.383,Z 779.752,A -85,B 0,C 180,E1 8263.813,E2 8263.813} C_VEL
LIN {X 0,Y 255.396,Z 799.055,A -85,B 0,C 180,E1 8262.777,E2 8262.777} C_VEL
LIN {X 0,Y 245.83,Z 818.52,A -85,B 0,C 180,E1 8261.369,E2 8261.369} C_VEL
LIN {X 0,Y 235.284,Z 837.188,A -85,B 0,C 180,E1 8259.581,E2 8259.581} C_VEL
LIN {X 0,Y 223.367,Z 855.797,A -85,B 0,C 180,E1 8257.226,E2 8257.226} C_VEL
LIN {X 0,Y 211.602,Z 872.285,A -85,B 0,C 180,E1 8254.48,E2 8254.48} C_VEL
LIN {X 0,Y 199.738,Z 887.429,A -85,B 0,C 180,E1 8251.158,E2 8251.158} C_VEL
LIN {X 0,Y 188.044,Z 901.3,A -85,B 0,C 180,E1 8247.145,E2 8247.145} C_VEL
LIN {X 0,Y 176.305,Z 914.617,A -85,B 0,C 180,E1 8242.021,E2 8242.021} C_VEL
LIN {X 0,Y 166.189,Z 925.939,A -85,B 0,C 180,E1 8236.213,E2 8236.213} C_VEL
LIN {X 0,Y 157.237,Z 936.312,A -85,B 0,C 180,E1 8229.013,E2 8229.013} C_VEL
LIN {X 0,Y 150.898,Z 944.629,A -85,B 0,C 180,E1 8221.118,E2 8221.118} C_VEL
LIN {X 0,Y 147.23,Z 951.23,A -85,B 0,C 180,E1 8212.545,E2 8212.545} C_VEL
LIN {X 0,Y 146.236,Z 955.597,A -85,B 0,C 180,E1 8204.654,E2 8204.654} C_VEL
LIN {X 0,Y 146.845,Z 958.09,A -85,B 0,C 180,E1 8197.434,E2 8197.434} C_VEL
LIN {X 0,Y 147.61,Z 959.002,A -85,B 0,C 180,E1 8192.33,E2 8192.33} C_VEL
LIN {X 0,Y 147.678,Z 959.068,A -85,B 0,C 180,E1 8188.45,E2 8188.45} C_VEL
LIN {X 0,Y 146.964,Z 958.278,A -85,B 0,C 180,E1 8183.354,E2 8183.354} C_VEL
LIN {X 0,Y 146.277,Z 956.213,A -85,B 0,C 180,E1 8176.966,E2 8176.966} C_VEL
LIN {X 0,Y 146.918,Z 952.061,A -85,B 0,C 180,E1 8168.803,E2 8168.803} C_VEL
LIN {X 0,Y 149.996,Z 946.019,A -85,B 0,C 180,E1 8160.449,E2 8160.449} C_VEL
LIN {X 0,Y 155.822,Z 937.963,A -85,B 0,C 180,E1 8152.447,E2 8152.447} C_VEL
LIN {X 0,Y 163.838,Z 928.474,A -85,B 0,C 180,E1 8145.435,E2 8145.435} C_VEL
LIN {X 0,Y 174.021,Z 917.067,A -85,B 0,C 180,E1 8139.144,E2 8139.144} C_VEL
LIN {X 0,Y 184.801,Z 904.98,A -85,B 0,C 180,E1 8134.137,E2 8134.137} C_VEL
LIN {X 0,Y 196.886,Z 890.734,A -85,B 0,C 180,E1 8129.739,E2 8129.739} C_VEL
LIN {X 0,Y 208.855,Z 875.653,A -85,B 0,C 180,E1 8126.22,E2 8126.22} C_VEL
LIN {X 0,Y 221.181,Z 858.775,A -85,B 0,C 180,E1 8123.246,E2 8123.246} C_VEL
LIN {X 0,Y 232.326,Z 841.874,A -85,B 0,C 180,E1 8120.966,E2 8120.966} C_VEL
LIN {X 0,Y 242.826,Z 823.794,A -85,B 0,C 180,E1 8119.112,E2 8119.112} C_VEL
LIN {X 0,Y 252.318,Z 805.187,A -85,B 0,C 180,E1 8117.652,E2 8117.652} C_VEL
LIN {X 0,Y 260.697,Z 786.225,A -85,B 0,C 180,E1 8116.52,E2 8116.52} C_VEL
LIN {X 0,Y 268.307,Z 765.403,A -85,B 0,C 180,E1 8115.592,E2 8115.592} C_VEL
LIN {X 0,Y 274.353,Z 744.215,A -85,B 0,C 180,E1 8114.856,E2 8114.856} C_VEL
LIN {X 0,Y 279.031,Z 721.677,A -85,B 0,C 180,E1 8114.236,E2 8114.236} C_VEL
LIN {X 0,Y 282.199,Z 697.387,A -85,B 0,C 180,E1 8113.713,E2 8113.713} C_VEL
LIN {X 0,Y 294.161,Z 580.497,A -85,B 0,C 180,E1 8111.424,E2 8111.424} C_VEL
LIN {X 0,Y 291.467,Z 573.272,A -85,B 0,C 180,E1 8108.383,E2 8108.383} C_VEL
LIN {X 0,Y 289.32,Z 567.464,A -85,B 0,C 180,E1 8105.155,E2 8105.155} C_VEL
LIN {X 0,Y 287.914,Z 563.605,A -85,B 0,C 180,E1 8101.99,E2 8101.99} C_VEL
LIN {X 0,Y 287.18,Z 560.649,A -85,B 0,C 180,E1 8098.204,E2 8098.204} C_VEL
LIN {X 0,Y 287.619,Z 560.539,A -85,B 0,C 180,E1 8093.412,E2 8093.412} C_VEL
LIN {X 0,Y 288.375,Z 561.418,A -85,B 0,C 180,E1 8091.224,E2 8091.224} C_VEL
LIN {X 0,Y 290.671,Z 565.652,A -85,B 0,C 180,E1 8087.08,E2 8087.08} C_VEL
LIN {X 0,Y 292.794,Z 569.716,A -85,B 0,C 180,E1 8084.45,E2 8084.45} C_VEL
LIN {X 0,Y 294.148,Z 572.543,A -85,B 0,C 180,E1 8083.019,E2 8083.019} C_VEL
LIN {X 0,Y 282.885,Z 685.408,A -85,B 0,C 180,E1 8080.868,E2 8080.868} C_VEL
LIN {X 0,Y 279.954,Z 706.724,A -85,B 0,C 180,E1 8080.236,E2 8080.236} C_VEL
LIN {X 0,Y 275.4,Z 727.956,A -85,B 0,C 180,E1 8079.376,E2 8079.376} C_VEL
LIN {X 0,Y 269.937,Z 746.85,A -85,B 0,C 180,E1 8078.374,E2 8078.374} C_VEL
LIN {X 0,Y 262.737,Z 766.697,A -85,B 0,C 180,E1 8077.049,E2 8077.049} C_VEL
LIN {X 0,Y 254.819,Z 784.7,A -85,B 0,C 180,E1 8075.535,E2 8075.535} C_VEL
LIN {X 0,Y 245.412,Z 802.635,A -85,B 0,C 180,E1 8073.634,E2 8073.634} C_VEL
LIN {X 0,Y 235.548,Z 818.75,A -85,B 0,C 180,E1 8071.471,E2 8071.471} C_VEL
LIN {X 0,Y 224.482,Z 834.586,A -85,B 0,C 180,E1 8068.768,E2 8068.768} C_VEL
LIN {X 0,Y 213.162,Z 848.871,A -85,B 0,C 180,E1 8065.634,E2 8065.634} C_VEL
LIN {X 0,Y 201.814,Z 861.709,A -85,B 0,C 180,E1 8061.966,E2 8061.966} C_VEL
LIN {X 0,Y 190.642,Z 873.014,A -85,B 0,C 180,E1 8057.681,E2 8057.681} C_VEL
LIN {X 0,Y 179.984,Z 882.899,A -85,B 0,C 180,E1 8052.661,E2 8052.661} C_VEL
LIN {X 0,Y 169.779,Z 891.714,A -85,B 0,C 180,E1 8046.493,E2 8046.493} C_VEL
LIN {X 0,Y 161.455,Z 898.55,A -85,B 0,C 180,E1 8039.693,E2 8039.693} C_VEL
LIN {X 0,Y 155.178,Z 903.609,A -85,B 0,C 180,E1 8032.339,E2 8032.339} C_VEL
LIN {X 0,Y 150.907,Z 907.109,A -85,B 0,C 180,E1 8024.188,E2 8024.188} C_VEL
LIN {X 0,Y 148.816,Z 908.858,A -85,B 0,C 180,E1 8016.169,E2 8016.169} C_VEL
LIN {X 0,Y 148.412,Z 909.231,A -85,B 0,C 180,E1 8008.068,E2 8008.068} C_VEL
LIN {X 0,Y 149.473,Z 908.356,A -85,B 0,C 180,E1 8000.373,E2 8000.373} C_VEL
LIN {X 0,Y 152.33,Z 905.933,A -85,B 0,C 180,E1 7992.427,E2 7992.427} C_VEL
LIN {X 0,Y 157.262,Z 901.955,A -85,B 0,C 180,E1 7984.789,E2 7984.789} C_VEL
LIN {X 0,Y 164.7,Z 895.986,A -85,B 0,C 180,E1 7977.298,E2 7977.298} C_VEL
LIN {X 0,Y 173.387,Z 888.802,A -85,B 0,C 180,E1 7971.059,E2 7971.059} C_VEL
LIN {X 0,Y 183.677,Z 879.753,A -85,B 0,C 180,E1 7965.399,E2 7965.399} C_VEL
LIN {X 0,Y 194.78,Z 869.106,A -85,B 0,C 180,E1 7960.565,E2 7960.565} C_VEL
LIN {X 0,Y 205.625,Z 857.671,A -85,B 0,C 180,E1 7956.654,E2 7956.654} C_VEL
LIN {X 0,Y 217.243,Z 844.131,A -85,B 0,C 180,E1 7953.114,E2 7953.114} C_VEL
LIN {X 0,Y 228.389,Z 829.542,A -85,B 0,C 180,E1 7950.168,E2 7950.168} C_VEL
LIN {X 0,Y 239.233,Z 813.375,A -85,B 0,C 180,E1 7947.63,E2 7947.63} C_VEL
LIN {X 0,Y 248.842,Z 796.73,A -85,B 0,C 180,E1 7945.581,E2 7945.581} C_VEL
LIN {X 0,Y 257.875,Z 778.499,A -85,B 0,C 180,E1 7943.799,E2 7943.799} C_VEL
LIN {X 0,Y 265.84,Z 759.242,A -85,B 0,C 180,E1 7942.308,E2 7942.308} C_VEL
LIN {X 0,Y 272.264,Z 740.205,A -85,B 0,C 180,E1 7941.139,E2 7941.139} C_VEL
LIN {X 0,Y 277.542,Z 719.767,A -85,B 0,C 180,E1 7940.162,E2 7940.162} C_VEL
LIN {X 0,Y 281.322,Z 699.332,A -85,B 0,C 180,E1 7939.422,E2 7939.422} C_VEL
LIN {X 0,Y 284.307,Z 673.133,A -85,B 0,C 180,E1 7938.749,E2 7938.749} C_VEL
LIN {X 0,Y 294.313,Z 572.445,A -85,B 0,C 180,E1 7936.835,E2 7936.835} C_VEL
LIN {X 0,Y 291.672,Z 567.368,A -85,B 0,C 180,E1 7933.885,E2 7933.885} C_VEL
LIN {X 0,Y 290.142,Z 564.533,A -85,B 0,C 180,E1 7931.732,E2 7931.732} C_VEL
LIN {X 0,Y 288.26,Z 561.058,A -85,B 0,C 180,E1 7927.775,E2 7927.775} C_VEL
LIN {X 0,Y 287.379,Z 560.573,A -85,B 0,C 180,E1 7923.391,E2 7923.391} C_VEL
LIN {X 0,Y 287.468,Z 561.201,A -85,B 0,C 180,E1 7921.196,E2 7921.196} C_VEL
LIN {X 0,Y 288.464,Z 564.744,A -85,B 0,C 180,E1 7917.12,E2 7917.12} C_VEL
LIN {X 0,Y 290.042,Z 569.125,A -85,B 0,C 180,E1 7913.965,E2 7913.965} C_VEL
LIN {X 0,Y 292.665,Z 576.053,A -85,B 0,C 180,E1 7910.413,E2 7910.413} C_VEL
LIN {X 0,Y 294.369,Z 580.977,A -85,B 0,C 180,E1 7908.536,E2 7908.536} C_VEL
LIN {X 0,Y 289.556,Z 627.457,A -85,B 0,C 180,E1 7907.661,E2 7907.661} C_VEL
LIN {X 0,Y 288.502,Z 635.147,A -85,B 0,C 180,E1 7907.703,E2 7907.703} C_VEL
LIN {X 0,Y 284.749,Z 655.659,A -85,B 0,C 180,E1 7908.52,E2 7908.52} C_VEL
LIN {X 0,Y 283.868,Z 662.26,A -85,B 0,C 180,E1 7908.543,E2 7908.543} C_VEL
LIN {X 0,Y 278.111,Z 714.581,A -85,B 0,C 180,E1 7907.523,E2 7907.523} C_VEL
LIN {X 0,Y 273.81,Z 737.133,A -85,B 0,C 180,E1 7906.962,E2 7906.962} C_VEL
LIN {X 0,Y 268.07,Z 758.32,A -85,B 0,C 180,E1 7906.297,E2 7906.297} C_VEL
LIN {X 0,Y 260.773,Z 779.203,A -85,B 0,C 180,E1 7905.479,E2 7905.479} C_VEL
LIN {X 0,Y 252.196,Z 799.309,A -85,B 0,C 180,E1 7904.432,E2 7904.432} C_VEL
LIN {X 0,Y 242.449,Z 818.631,A -85,B 0,C 180,E1 7903.075,E2 7903.075} C_VEL
LIN {X 0,Y 231.671,Z 837.066,A -85,B 0,C 180,E1 7901.346,E2 7901.346} C_VEL
LIN {X 0,Y 219.844,Z 854.931,A -85,B 0,C 180,E1 7899.137,E2 7899.137} C_VEL
LIN {X 0,Y 207.693,Z 871.386,A -85,B 0,C 180,E1 7896.449,E2 7896.449} C_VEL
LIN {X 0,Y 195.079,Z 886.88,A -85,B 0,C 180,E1 7893.093,E2 7893.093} C_VEL
LIN {X 0,Y 182.237,Z 901.381,A -85,B 0,C 180,E1 7888.853,E2 7888.853} C_VEL
LIN {X 0,Y 170.62,Z 913.818,A -85,B 0,C 180,E1 7883.963,E2 7883.963} C_VEL
LIN {X 0,Y 159.787,Z 925.181,A -85,B 0,C 180,E1 7877.969,E2 7877.969} C_VEL
LIN {X 0,Y 150.374,Z 935.344,A -85,B 0,C 180,E1 7870.66,E2 7870.66} C_VEL
LIN {X 0,Y 143.508,Z 943.575,A -85,B 0,C 180,E1 7862.442,E2 7862.442} C_VEL
LIN {X 0,Y 139.525,Z 949.95,A -85,B 0,C 180,E1 7853.659,E2 7853.659} C_VEL
LIN {X 0,Y 138.31,Z 954.377,A -85,B 0,C 180,E1 7845.085,E2 7845.085} C_VEL
LIN {X 0,Y 138.864,Z 956.735,A -85,B 0,C 180,E1 7837.864,E2 7837.864} C_VEL
LIN {X 0,Y 139.694,Z 957.668,A -85,B 0,C 180,E1 7832.463,E2 7832.463} C_VEL
LIN {X 0,Y 139.775,Z 957.737,A -85,B 0,C 180,E1 7828.362,E2 7828.362} C_VEL
LIN {X 0,Y 138.983,Z 956.926,A -85,B 0,C 180,E1 7822.977,E2 7822.977} C_VEL
LIN {X 0,Y 138.314,Z 954.835,A -85,B 0,C 180,E1 7816.202,E2 7816.202} C_VEL
LIN {X 0,Y 139.296,Z 950.437,A -85,B 0,C 180,E1 7807.198,E2 7807.198} C_VEL
LIN {X 0,Y 142.84,Z 944.487,A -85,B 0,C 180,E1 7798.646,E2 7798.646} C_VEL
LIN {X 0,Y 149.337,Z 936.405,A -85,B 0,C 180,E1 7790.349,E2 7790.349} C_VEL
LIN {X 0,Y 157.919,Z 927.04,A -85,B 0,C 180,E1 7783.279,E2 7783.279} C_VEL
LIN {X 0,Y 168.815,Z 915.627,A -85,B 0,C 180,E1 7776.92,E2 7776.92} C_VEL
LIN {X 0,Y 180.753,Z 902.917,A -85,B 0,C 180,E1 7771.701,E2 7771.701} C_VEL
LIN {X 0,Y 193.588,Z 888.452,A -85,B 0,C 180,E1 7767.346,E2 7767.346} C_VEL
LIN {X 0,Y 206.151,Z 873.118,A -85,B 0,C 180,E1 7763.916,E2 7763.916} C_VEL
LIN {X 0,Y 218.618,Z 856.44,A -85,B 0,C 180,E1 7761.109,E2 7761.109} C_VEL
LIN {X 0,Y 229.914,Z 839.659,A -85,B 0,C 180,E1 7758.957,E2 7758.957} C_VEL
LIN {X 0,Y 241.097,Z 820.776,A -85,B 0,C 180,E1 7757.124,E2 7757.124} C_VEL
LIN {X 0,Y 250.717,Z 801.985,A -85,B 0,C 180,E1 7755.756,E2 7755.756} C_VEL
LIN {X 0,Y 259.852,Z 781.044,A -85,B 0,C 180,E1 7754.623,E2 7754.623} C_VEL
LIN {X 0,Y 267.145,Z 760.719,A -85,B 0,C 180,E1 7753.8,E2 7753.8} C_VEL
LIN {X 0,Y 273.284,Z 738.618,A -85,B 0,C 180,E1 7753.091,E2 7753.091} C_VEL
LIN {X 0,Y 277.639,Z 716.13,A -85,B 0,C 180,E1 7752.525,E2 7752.525} C_VEL
LIN {X 0,Y 281.818,Z 680.008,A -85,B 0,C 180,E1 7751.81,E2 7751.81} C_VEL
LIN {X 0,Y 291.718,Z 585.614,A -85,B 0,C 180,E1 7750.017,E2 7750.017} C_VEL
LIN {X 0,Y 289.488,Z 579.308,A -85,B 0,C 180,E1 7747.142,E2 7747.142} C_VEL
LIN {X 0,Y 287.878,Z 574.648,A -85,B 0,C 180,E1 7744.382,E2 7744.382} C_VEL
LIN {X 0,Y 286.792,Z 571.322,A -85,B 0,C 180,E1 7741.598,E2 7741.598} C_VEL
LIN {X 0,Y 286.188,Z 568.552,A -85,B 0,C 180,E1 7737.997,E2 7737.997} C_VEL
LIN {X 0,Y 286.652,Z 568.494,A -85,B 0,C 180,E1 7733.39,E2 7733.39} C_VEL
LIN {X 0,Y 287.33,Z 569.322,A -85,B 0,C 180,E1 7731.394,E2 7731.394} C_VEL
LIN {X 0,Y 289.426,Z 573.359,A -85,B 0,C 180,E1 7727.429,E2 7727.429} C_VEL
LIN {X 0,Y 291.463,Z 577.45,A -85,B 0,C 180,E1 7724.785,E2 7724.785} C_VEL
LIN {X 0,Y 291.735,Z 578.32,A -85,B 0,C 180,E1 7724.442,E2 7724.442} C_VEL
LIN {X 0,Y 280.714,Z 685.937,A -85,B 0,C 180,E1 7722.43,E2 7722.43} C_VEL
LIN {X 0,Y 277.692,Z 707.492,A -85,B 0,C 180,E1 7721.805,E2 7721.805} C_VEL
LIN {X 0,Y 273.017,Z 728.792,A -85,B 0,C 180,E1 7720.963,E2 7720.963} C_VEL
LIN {X 0,Y 267.15,Z 748.578,A -85,B 0,C 180,E1 7719.935,E2 7719.935} C_VEL
LIN {X 0,Y 259.778,Z 768.286,A -85,B 0,C 180,E1 7718.642,E2 7718.642} C_VEL
LIN {X 0,Y 251.452,Z 786.617,A -85,B 0,C 180,E1 7717.124,E2 7717.124} C_VEL
LIN {X 0,Y 241.675,Z 804.721,A -85,B 0,C 180,E1 7715.232,E2 7715.232} C_VEL
LIN {X 0,Y 231.119,Z 821.338,A -85,B 0,C 180,E1 7713.01,E2 7713.01} C_VEL
LIN {X 0,Y 220.495,Z 835.976,A -85,B 0,C 180,E1 7710.522,E2 7710.522} C_VEL
LIN {X 0,Y 208.803,Z 850.242,A -85,B 0,C 180,E1 7707.424,E2 7707.424} C_VEL
LIN {X 0,Y 197.034,Z 863.067,A -85,B 0,C 180,E1 7703.78,E2 7703.78} C_VEL
LIN {X 0,Y 184.784,Z 874.961,A -85,B 0,C 180,E1 7699.239,E2 7699.239} C_VEL
LIN {X 0,Y 173.681,Z 884.721,A -85,B 0,C 180,E1 7694.146,E2 7694.146} C_VEL
LIN {X 0,Y 163.464,Z 893.055,A -85,B 0,C 180,E1 7688.149,E2 7688.149} C_VEL
LIN {X 0,Y 154.604,Z 899.888,A -85,B 0,C 180,E1 7681.151,E2 7681.151} C_VEL
LIN {X 0,Y 147.872,Z 904.945,A -85,B 0,C 180,E1 7673.508,E2 7673.508} C_VEL
LIN {X 0,Y 143.245,Z 908.443,A -85,B 0,C 180,E1 7664.964,E2 7664.964} C_VEL
LIN {X 0,Y 140.968,Z 910.188,A -85,B 0,C 180,E1 7656.514,E2 7656.514} C_VEL
LIN {X 0,Y 140.515,Z 910.578,A -85,B 0,C 180,E1 7648.368,E2 7648.368} C_VEL
LIN {X 0,Y 141.587,Z 909.763,A -85,B 0,C 180,E1 7640.242,E2 7640.242} C_VEL
LIN {X 0,Y 144.596,Z 907.404,A -85,B 0,C 180,E1 7631.871,E2 7631.871} C_VEL
LIN {X 0,Y 149.814,Z 903.517,A -85,B 0,C 180,E1 7623.867,E2 7623.867} C_VEL
LIN {X 0,Y 157.315,Z 897.917,A -85,B 0,C 180,E1 7616.369,E2 7616.369} C_VEL
LIN {X 0,Y 166.293,Z 890.984,A -85,B 0,C 180,E1 7609.961,E2 7609.961} C_VEL
LIN {X 0,Y 176.96,Z 882.065,A -85,B 0,C 180,E1 7604.15,E2 7604.15} C_VEL
LIN {X 0,Y 187.808,Z 872.235,A -85,B 0,C 180,E1 7599.476,E2 7599.476} C_VEL
LIN {X 0,Y 200.316,Z 859.755,A -85,B 0,C 180,E1 7595.063,E2 7595.063} C_VEL
LIN {X 0,Y 211.584,Z 847.263,A -85,B 0,C 180,E1 7591.73,E2 7591.73} C_VEL
LIN {X 0,Y 223.401,Z 832.49,A -85,B 0,C 180,E1 7588.7,E2 7588.7} C_VEL
LIN {X 0,Y 234.507,Z 816.542,A -85,B 0,C 180,E1 7586.179,E2 7586.179} C_VEL
LIN {X 0,Y 244.709,Z 799.676,A -85,B 0,C 180,E1 7584.088,E2 7584.088} C_VEL
LIN {X 0,Y 253.998,Z 781.767,A -85,B 0,C 180,E1 7582.333,E2 7582.333} C_VEL
LIN {X 0,Y 262.148,Z 763.073,A -85,B 0,C 180,E1 7580.873,E2 7580.873} C_VEL
LIN {X 0,Y 269.124,Z 743.236,A -85,B 0,C 180,E1 7579.656,E2 7579.656} C_VEL
LIN {X 0,Y 274.571,Z 723.238,A -85,B 0,C 180,E1 7578.694,E2 7578.694} C_VEL
LIN {X 0,Y 278.824,Z 701.76,A -85,B 0,C 180,E1 7577.909,E2 7577.909} C_VEL
LIN {X 0,Y 281.683,Z 678.686,A -85,B 0,C 180,E1 7577.301,E2 7577.301} C_VEL
LIN {X 0,Y 291.949,Z 578.194,A -85,B 0,C 180,E1 7575.443,E2 7575.443} C_VEL
LIN {X 0,Y 290.031,Z 574.394,A -85,B 0,C 180,E1 7573.051,E2 7573.051} C_VEL
LIN {X 0,Y 288.805,Z 572.075,A -85,B 0,C 180,E1 7571.179,E2 7571.179} C_VEL
LIN {X 0,Y 287.219,Z 568.958,A -85,B 0,C 180,E1 7567.602,E2 7567.602} C_VEL
LIN {X 0,Y 286.403,Z 568.514,A -85,B 0,C 180,E1 7563.403,E2 7563.403} C_VEL
LIN {X 0,Y 286.458,Z 569.077,A -85,B 0,C 180,E1 7561.401,E2 7561.401} C_VEL
LIN {X 0,Y 287.341,Z 572.553,A -85,B 0,C 180,E1 7557.408,E2 7557.408} C_VEL
LIN {X 0,Y 288.778,Z 576.806,A -85,B 0,C 180,E1 7554.337,E2 7554.337} C_VEL
LIN {X 0,Y 291.113,Z 583.409,A -85,B 0,C 180,E1 7550.96,E2 7550.96} C_VEL
LIN {X 0,Y 291.919,Z 585.999,A -85,B 0,C 180,E1 7549.963,E2 7549.963} C_VEL
LIN {X 0,Y 283.868,Z 662.26,A -85,B 0,C 180,E1 7548.543,E2 7548.543} C_VEL
LIN {X 0,Y 282.82,Z 669.948,A -85,B 0,C 180,E1 7548.589,E2 7548.589} C_VEL
LIN {X 0,Y 279.159,Z 690.462,A -85,B 0,C 180,E1 7549.432,E2 7549.432} C_VEL
LIN {X 0,Y 278.268,Z 697.064,A -85,B 0,C 180,E1 7549.47,E2 7549.47} C_VEL
LIN {X 0,Y 275.056,Z 720.165,A -85,B 0,C 180,E1 7548.998,E2 7548.998} C_VEL
LIN {X 0,Y 270.069,Z 743.055,A -85,B 0,C 180,E1 7548.412,E2 7548.412} C_VEL
LIN {X 0,Y 263.907,Z 763.772,A -85,B 0,C 180,E1 7547.751,E2 7547.751} C_VEL
LIN {X 0,Y 255.968,Z 784.724,A -85,B 0,C 180,E1 7546.906,E2 7546.906} C_VEL
LIN {X 0,Y 246.945,Z 804.189,A -85,B 0,C 180,E1 7545.843,E2 7545.843} C_VEL
LIN {X 0,Y 236.616,Z 823.294,A -85,B 0,C 180,E1 7544.444,E2 7544.444} C_VEL
LIN {X 0,Y 225.2,Z 841.685,A -85,B 0,C 180,E1 7542.648,E2 7542.648} C_VEL
LIN {X 0,Y 213.249,Z 858.681,A -85,B 0,C 180,E1 7540.449,E2 7540.449} C_VEL
LIN {X 0,Y 200.493,Z 874.79,A -85,B 0,C 180,E1 7537.67,E2 7537.67} C_VEL
LIN {X 0,Y 187.6,Z 889.643,A -85,B 0,C 180,E1 7534.244,E2 7534.244} C_VEL
LIN {X 0,Y 175.194,Z 902.91,A -85,B 0,C 180,E1 7530.16,E2 7530.16} C_VEL
LIN {X 0,Y 162.635,Z 915.56,A -85,B 0,C 180,E1 7524.846,E2 7524.846} C_VEL
LIN {X 0,Y 151.722,Z 926.21,A -85,B 0,C 180,E1 7518.696,E2 7518.696} C_VEL
LIN {X 0,Y 142.002,Z 936.001,A -85,B 0,C 180,E1 7510.903,E2 7510.903} C_VEL
LIN {X 0,Y 135.38,Z 943.546,A -85,B 0,C 180,E1 7502.624,E2 7502.624} C_VEL
LIN {X 0,Y 131.535,Z 949.331,A -85,B 0,C 180,E1 7493.757,E2 7493.757} C_VEL
LIN {X 0,Y 130.374,Z 953.476,A -85,B 0,C 180,E1 7484.66,E2 7484.66} C_VEL
LIN {X 0,Y 131.025,Z 955.63,A -85,B 0,C 180,E1 7477.246,E2 7477.246} C_VEL
LIN {X 0,Y 131.867,Z 956.409,A -85,B 0,C 180,E1 7471.739,E2 7471.739} C_VEL
LIN {X 0,Y 131.823,Z 956.369,A -85,B 0,C 180,E1 7467.828,E2 7467.828} C_VEL
LIN {X 0,Y 130.937,Z 955.469,A -85,B 0,C 180,E1 7462.102,E2 7462.102} C_VEL
LIN {X 0,Y 130.388,Z 953.136,A -85,B 0,C 180,E1 7454.435,E2 7454.435} C_VEL
LIN {X 0,Y 131.798,Z 948.773,A -85,B 0,C 180,E1 7445.344,E2 7445.344} C_VEL
LIN {X 0,Y 136.202,Z 942.472,A -85,B 0,C 180,E1 7436.094,E2 7436.094} C_VEL
LIN {X 0,Y 143.644,Z 934.284,A -85,B 0,C 180,E1 7427.538,E2 7427.538} C_VEL
LIN {X 0,Y 153.513,Z 924.37,A -85,B 0,C 180,E1 7420.15,E2 7420.15} C_VEL
LIN {X 0,Y 165.136,Z 912.914,A -85,B 0,C 180,E1 7413.963,E2 7413.963} C_VEL
LIN {X 0,Y 178.017,Z 899.812,A -85,B 0,C 180,E1 7408.826,E2 7408.826} C_VEL
LIN {X 0,Y 191.131,Z 885.596,A -85,B 0,C 180,E1 7404.739,E2 7404.739} C_VEL
LIN {X 0,Y 204.536,Z 869.688,A -85,B 0,C 180,E1 7401.388,E2 7401.388} C_VEL
LIN {X 0,Y 216.913,Z 853.359,A -85,B 0,C 180,E1 7398.823,E2 7398.823} C_VEL
LIN {X 0,Y 229.102,Z 835.353,A -85,B 0,C 180,E1 7396.696,E2 7396.696} C_VEL
LIN {X 0,Y 240.168,Z 816.736,A -85,B 0,C 180,E1 7395.041,E2 7395.041} C_VEL
LIN {X 0,Y 250.11,Z 797.341,A -85,B 0,C 180,E1 7393.755,E2 7393.755} C_VEL
LIN {X 0,Y 258.837,Z 777.022,A -85,B 0,C 180,E1 7392.77,E2 7392.77} C_VEL
LIN {X 0,Y 266.105,Z 756.26,A -85,B 0,C 180,E1 7392.006,E2 7392.006} C_VEL
LIN {X 0,Y 271.953,Z 734.547,A -85,B 0,C 180,E1 7391.366,E2 7391.366} C_VEL
LIN {X 0,Y 276.163,Z 712.353,A -85,B 0,C 180,E1 7390.84,E2 7390.84} C_VEL
LIN {X 0,Y 289.415,Z 590.72,A -85,B 0,C 180,E1 7388.543,E2 7388.543} C_VEL
LIN {X 0,Y 287.312,Z 584.309,A -85,B 0,C 180,E1 7385.291,E2 7385.291} C_VEL
LIN {X 0,Y 285.863,Z 579.503,A -85,B 0,C 180,E1 7381.803,E2 7381.803} C_VEL
LIN {X 0,Y 285.199,Z 576.458,A -85,B 0,C 180,E1 7377.789,E2 7377.789} C_VEL
LIN {X 0,Y 285.682,Z 576.448,A -85,B 0,C 180,E1 7373.367,E2 7373.367} C_VEL
LIN {X 0,Y 286.279,Z 577.224,A -85,B 0,C 180,E1 7371.564,E2 7371.564} C_VEL
LIN {X 0,Y 288.191,Z 581.067,A -85,B 0,C 180,E1 7367.781,E2 7367.781} C_VEL
LIN {X 0,Y 289.51,Z 583.989,A -85,B 0,C 180,E1 7365.89,E2 7365.89} C_VEL
LIN {X 0,Y 278.718,Z 686.785,A -85,B 0,C 180,E1 7364.008,E2 7364.008} C_VEL
LIN {X 0,Y 275.614,Z 708.382,A -85,B 0,C 180,E1 7363.395,E2 7363.395} C_VEL
LIN {X 0,Y 270.833,Z 729.684,A -85,B 0,C 180,E1 7362.574,E2 7362.574} C_VEL
LIN {X 0,Y 264.984,Z 749.059,A -85,B 0,C 180,E1 7361.599,E2 7361.599} C_VEL
LIN {X 0,Y 257.442,Z 768.901,A -85,B 0,C 180,E1 7360.342,E2 7360.342} C_VEL
LIN {X 0,Y 249.137,Z 786.919,A -85,B 0,C 180,E1 7358.904,E2 7358.904} C_VEL
LIN {X 0,Y 239.295,Z 804.785,A -85,B 0,C 180,E1 7357.105,E2 7357.105} C_VEL
LIN {X 0,Y 228.721,Z 821.188,A -85,B 0,C 180,E1 7355.003,E2 7355.003} C_VEL
LIN {X 0,Y 217.49,Z 836.401,A -85,B 0,C 180,E1 7352.519,E2 7352.519} C_VEL
LIN {X 0,Y 206.143,Z 850.009,A -85,B 0,C 180,E1 7349.684,E2 7349.684} C_VEL
LIN {X 0,Y 193.857,Z 863.006,A -85,B 0,C 180,E1 7346.129,E2 7346.129} C_VEL
LIN {X 0,Y 181.651,Z 874.533,A -85,B 0,C 180,E1 7341.907,E2 7341.907} C_VEL
LIN {X 0,Y 169.827,Z 884.64,A -85,B 0,C 180,E1 7336.883,E2 7336.883} C_VEL
LIN {X 0,Y 158.814,Z 893.286,A -85,B 0,C 180,E1 7330.895,E2 7330.895} C_VEL
LIN {X 0,Y 149.501,Z 900.127,A -85,B 0,C 180,E1 7324.174,E2 7324.174} C_VEL
LIN {X 0,Y 141.828,Z 905.431,A -85,B 0,C 180,E1 7316.364,E2 7316.364} C_VEL
LIN {X 0,Y 136.511,Z 909.083,A -85,B 0,C 180,E1 7307.913,E2 7307.913} C_VEL
LIN {X 0,Y 133.522,Z 911.231,A -85,B 0,C 180,E1 7299.045,E2 7299.045} C_VEL
LIN {X 0,Y 132.611,Z 911.958,A -85,B 0,C 180,E1 7290.43,E2 7290.43} C_VEL
LIN {X 0,Y 133.334,Z 911.373,A -85,B 0,C 180,E1 7281.808,E2 7281.808} C_VEL
LIN {X 0,Y 136.107,Z 909.425,A -85,B 0,C 180,E1 7272.912,E2 7272.912} C_VEL
LIN {X 0,Y 141.178,Z 905.982,A -85,B 0,C 180,E1 7264.405,E2 7264.405} C_VEL
LIN {X 0,Y 149.018,Z 900.529,A -85,B 0,C 180,E1 7256.161,E2 7256.161} C_VEL
LIN {X 0,Y 158.615,Z 893.532,A -85,B 0,C 180,E1 7249.153,E2 7249.153} C_VEL
LIN {X 0,Y 169.741,Z 884.836,A -85,B 0,C 180,E1 7243.083,E2 7243.083} C_VEL
LIN {X 0,Y 182.215,Z 874.177,A -85,B 0,C 180,E1 7237.805,E2 7237.805} C_VEL
LIN {X 0,Y 194.466,Z 862.567,A -85,B 0,C 180,E1 7233.606,E2 7233.606} C_VEL
LIN {X 0,Y 206.795,Z 849.51,A -85,B 0,C 180,E1 7230.072,E2 7230.072} C_VEL
LIN {X 0,Y 218.944,Z 834.84,A -85,B 0,C 180,E1 7227.072,E2 7227.072} C_VEL
LIN {X 0,Y 229.941,Z 819.706,A -85,B 0,C 180,E1 7224.67,E2 7224.67} C_VEL
LIN {X 0,Y 240.83,Z 802.481,A -85,B 0,C 180,E1 7222.53,E2 7222.53} C_VEL
LIN {X 0,Y 250.294,Z 785.035,A -85,B 0,C 180,E1 7220.822,E2 7220.822} C_VEL
LIN {X 0,Y 258.617,Z 766.685,A -85,B 0,C 180,E1 7219.393,E2 7219.393} C_VEL
LIN {X 0,Y 265.584,Z 747.929,A -85,B 0,C 180,E1 7218.233,E2 7218.233} C_VEL
LIN {X 0,Y 271.804,Z 726.633,A -85,B 0,C 180,E1 7217.193,E2 7217.193} C_VEL
LIN {X 0,Y 276.244,Z 705.921,A -85,B 0,C 180,E1 7216.424,E2 7216.424} C_VEL
LIN {X 0,Y 279.246,Z 684.222,A -85,B 0,C 180,E1 7215.829,E2 7215.829} C_VEL
LIN {X 0,Y 289.718,Z 583.944,A -85,B 0,C 180,E1 7213.98,E2 7213.98} C_VEL
LIN {X 0,Y 287.723,Z 579.975,A -85,B 0,C 180,E1 7211.019,E2 7211.019} C_VEL
LIN {X 0,Y 286.181,Z 576.86,A -85,B 0,C 180,E1 7207.428,E2 7207.428} C_VEL
LIN {X 0,Y 285.428,Z 576.459,A -85,B 0,C 180,E1 7203.371,E2 7203.371} C_VEL
LIN {X 0,Y 285.453,Z 576.954,A -85,B 0,C 180,E1 7201.606,E2 7201.606} C_VEL
LIN {X 0,Y 286.226,Z 580.361,A -85,B 0,C 180,E1 7197.698,E2 7197.698} C_VEL
LIN {X 0,Y 287.64,Z 584.797,A -85,B 0,C 180,E1 7194.515,E2 7194.515} C_VEL
LIN {X 0,Y 289.654,Z 590.996,A -85,B 0,C 180,E1 7191.418,E2 7191.418} C_VEL
LIN {X 0,Y 278.268,Z 697.064,A -85,B 0,C 180,E1 7189.47,E2 7189.47} C_VEL
LIN {X 0,Y 277.131,Z 704.744,A -85,B 0,C 180,E1 7189.543,E2 7189.543} C_VEL
LIN {X 0,Y 272.701,Z 723.987,A -85,B 0,C 180,E1 7190.359,E2 7190.359} C_VEL
LIN {X 0,Y 270.847,Z 731.539,A -85,B 0,C 180,E1 7190.36,E2 7190.36} C_VEL
LIN {X 0,Y 264.918,Z 753.801,A -85,B 0,C 180,E1 7189.75,E2 7189.75} C_VEL
LIN {X 0,Y 257.626,Z 774.691,A -85,B 0,C 180,E1 7189.038,E2 7189.038} C_VEL
LIN {X 0,Y 248.77,Z 795.177,A -85,B 0,C 180,E1 7188.124,E2 7188.124} C_VEL
LIN {X 0,Y 238.658,Z 814.63,A -85,B 0,C 180,E1 7186.925,E2 7186.925} C_VEL
LIN {X 0,Y 227.327,Z 833.422,A -85,B 0,C 180,E1 7185.364,E2 7185.364} C_VEL
LIN {X 0,Y 214.942,Z 851.365,A -85,B 0,C 180,E1 7183.372,E2 7183.372} C_VEL
LIN {X 0,Y 202.072,Z 867.921,A -85,B 0,C 180,E1 7180.908,E2 7180.908} C_VEL
LIN {X 0,Y 188.074,Z 883.972,A -85,B 0,C 180,E1 7177.662,E2 7177.662} C_VEL
LIN {X 0,Y 174.874,Z 897.739,A -85,B 0,C 180,E1 7173.843,E2 7173.843} C_VEL
LIN {X 0,Y 161.251,Z 910.945,A -85,B 0,C 180,E1 7168.828,E2 7168.828} C_VEL
LIN {X 0,Y 149.147,Z 922.191,A -85,B 0,C 180,E1 7162.891,E2 7162.891} C_VEL
LIN {X 0,Y 138.003,Z 932.495,A -85,B 0,C 180,E1 7155.234,E2 7155.234} C_VEL
LIN {X 0,Y 129.634,Z 940.741,A -85,B 0,C 180,E1 7146.431,E2 7146.431} C_VEL
LIN {X 0,Y 124.436,Z 947.143,A -85,B 0,C 180,E1 7136.74,E2 7136.74} C_VEL
LIN {X 0,Y 122.485,Z 951.773,A -85,B 0,C 180,E1 7126.601,E2 7126.601} C_VEL
LIN {X 0,Y 122.938,Z 954.12,A -85,B 0,C 180,E1 7118.419,E2 7118.419} C_VEL
LIN {X 0,Y 123.955,Z 955.076,A -85,B 0,C 180,E1 7111.85,E2 7111.85} C_VEL
LIN {X 0,Y 123.956,Z 955.072,A -85,B 0,C 180,E1 7108.153,E2 7108.153} C_VEL
LIN {X 0,Y 123.005,Z 954.213,A -85,B 0,C 180,E1 7102.06,E2 7102.06} C_VEL
LIN {X 0,Y 122.468,Z 951.913,A -85,B 0,C 180,E1 7093.887,E2 7093.887} C_VEL
LIN {X 0,Y 124.272,Z 947.369,A -85,B 0,C 180,E1 7083.74,E2 7083.74} C_VEL
LIN {X 0,Y 129.309,Z 941.053,A -85,B 0,C 180,E1 7074.015,E2 7074.015} C_VEL
LIN {X 0,Y 137.532,Z 932.859,A -85,B 0,C 180,E1 7065.163,E2 7065.163} C_VEL
LIN {X 0,Y 147.987,Z 923.133,A -85,B 0,C 180,E1 7057.777,E2 7057.777} C_VEL
LIN {X 0,Y 160.565,Z 911.474,A -85,B 0,C 180,E1 7051.46,E2 7051.46} C_VEL
LIN {X 0,Y 174.114,Z 898.366,A -85,B 0,C 180,E1 7046.398,E2 7046.398} C_VEL
LIN {X 0,Y 187.264,Z 884.709,A -85,B 0,C 180,E1 7042.544,E2 7042.544} C_VEL
LIN {X 0,Y 200.798,Z 869.211,A -85,B 0,C 180,E1 7039.354,E2 7039.354} C_VEL
LIN {X 0,Y 213.461,Z 853.1,A -85,B 0,C 180,E1 7036.882,E2 7036.882} C_VEL
LIN {X 0,Y 225.971,Z 835.225,A -85,B 0,C 180,E1 7034.83,E2 7034.83} C_VEL
LIN {X 0,Y 237.255,Z 816.839,A -85,B 0,C 180,E1 7033.248,E2 7033.248} C_VEL
LIN {X 0,Y 247.828,Z 796.66,A -85,B 0,C 180,E1 7031.972,E2 7031.972} C_VEL
LIN {X 0,Y 256.691,Z 776.461,A -85,B 0,C 180,E1 7031.046,E2 7031.046} C_VEL
LIN {X 0,Y 264.201,Z 755.411,A -85,B 0,C 180,E1 7030.312,E2 7030.312} C_VEL
LIN {X 0,Y 270.083,Z 734.013,A -85,B 0,C 180,E1 7029.711,E2 7029.711} C_VEL
LIN {X 0,Y 274.408,Z 711.778,A -85,B 0,C 180,E1 7029.204,E2 7029.204} C_VEL
LIN {X 0,Y 286.962,Z 599.543,A -85,B 0,C 180,E1 7027.18,E2 7027.18} C_VEL
LIN {X 0,Y 287.329,Z 596.11,A -85,B 0,C 180,E1 7027.106,E2 7027.106} C_VEL
LIN {X 0,Y 285.615,Z 590.371,A -85,B 0,C 180,E1 7023.914,E2 7023.914} C_VEL
LIN {X 0,Y 284.627,Z 586.909,A -85,B 0,C 180,E1 7021.006,E2 7021.006} C_VEL
LIN {X 0,Y 284.224,Z 584.403,A -85,B 0,C 180,E1 7017.782,E2 7017.782} C_VEL
LIN {X 0,Y 284.658,Z 584.35,A -85,B 0,C 180,E1 7013.546,E2 7013.546} C_VEL
LIN {X 0,Y 285.228,Z 585.126,A -85,B 0,C 180,E1 7011.736,E2 7011.736} C_VEL
LIN {X 0,Y 287.023,Z 588.917,A -85,B 0,C 180,E1 7008.037,E2 7008.037} C_VEL
LIN {X 0,Y 287.434,Z 590.065,A -85,B 0,C 180,E1 7007.353,E2 7007.353} C_VEL
LIN {X 0,Y 276.949,Z 687.522,A -85,B 0,C 180,E1 7005.61,E2 7005.61} C_VEL
LIN {X 0,Y 273.767,Z 709.185,A -85,B 0,C 180,E1 7005.01,E2 7005.01} C_VEL
LIN {X 0,Y 268.914,Z 730.384,A -85,B 0,C 180,E1 7004.218,E2 7004.218} C_VEL
LIN {X 0,Y 262.748,Z 750.402,A -85,B 0,C 180,E1 7003.242,E2 7003.242} C_VEL
LIN {X 0,Y 254.829,Z 770.673,A -85,B 0,C 180,E1 7001.99,E2 7001.99} C_VEL
LIN {X 0,Y 245.994,Z 789.201,A -85,B 0,C 180,E1 7000.539,E2 7000.539} C_VEL
LIN {X 0,Y 235.932,Z 806.957,A -85,B 0,C 180,E1 6998.785,E2 6998.785} C_VEL
LIN {X 0,Y 224.845,Z 823.557,A -85,B 0,C 180,E1 6996.685,E2 6996.685} C_VEL
LIN {X 0,Y 213.172,Z 838.759,A -85,B 0,C 180,E1 6994.217,E2 6994.217} C_VEL
LIN {X 0,Y 200.735,Z 852.98,A -85,B 0,C 180,E1 6991.229,E2 6991.229} C_VEL
LIN {X 0,Y 188.113,Z 865.777,A -85,B 0,C 180,E1 6987.674,E2 6987.674} C_VEL
LIN {X 0,Y 174.85,Z 877.668,A -85,B 0,C 180,E1 6983.175,E2 6983.175} C_VEL
LIN {X 0,Y 162.669,Z 887.413,A -85,B 0,C 180,E1 6978.042,E2 6978.042} C_VEL
LIN {X 0,Y 151.295,Z 895.738,A -85,B 0,C 180,E1 6971.866,E2 6971.866} C_VEL
LIN {X 0,Y 141.249,Z 902.566,A -85,B 0,C 180,E1 6964.487,E2 6964.487} C_VEL
LIN {X 0,Y 133.474,Z 907.615,A -85,B 0,C 180,E1 6956.225,E2 6956.225} C_VEL
LIN {X 0,Y 128.013,Z 911.11,A -85,B 0,C 180,E1 6946.794,E2 6946.794} C_VEL
LIN {X 0,Y 125.29,Z 912.847,A -85,B 0,C 180,E1 6937.334,E2 6937.334} C_VEL
LIN {X 0,Y 124.742,Z 913.234,A -85,B 0,C 180,E1 6928.161,E2 6928.161} C_VEL
LIN {X 0,Y 126.038,Z 912.423,A -85,B 0,C 180,E1 6919.024,E2 6919.024} C_VEL
LIN {X 0,Y 129.623,Z 910.071,A -85,B 0,C 180,E1 6909.69,E2 6909.69} C_VEL
LIN {X 0,Y 135.745,Z 906.188,A -85,B 0,C 180,E1 6900.914,E2 6900.914} C_VEL
LIN {X 0,Y 144.29,Z 900.641,A -85,B 0,C 180,E1 6892.927,E2 6892.927} C_VEL
LIN {X 0,Y 154.474,Z 893.664,A -85,B 0,C 180,E1 6886.17,E2 6886.17} C_VEL
LIN {X 0,Y 166.296,Z 884.749,A -85,B 0,C 180,E1 6880.223,E2 6880.223} C_VEL
LIN {X 0,Y 178.841,Z 874.338,A -85,B 0,C 180,E1 6875.295,E2 6875.295} C_VEL
LIN {X 0,Y 191.662,Z 862.473,A -85,B 0,C 180,E1 6871.187,E2 6871.187} C_VEL
LIN {X 0,Y 203.718,Z 850.014,A -85,B 0,C 180,E1 6867.948,E2 6867.948} C_VEL
LIN {X 0,Y 216.265,Z 835.257,A -85,B 0,C 180,E1 6865.029,E2 6865.029} C_VEL
LIN {X 0,Y 227.584,Z 819.954,A -85,B 0,C 180,E1 6862.702,E2 6862.702} C_VEL
LIN {X 0,Y 238.804,Z 802.455,A -85,B 0,C 180,E1 6860.624,E2 6860.624} C_VEL
LIN {X 0,Y 248.455,Z 784.824,A -85,B 0,C 180,E1 6858.98,E2 6858.98} C_VEL
LIN {X 0,Y 256.978,Z 766.309,A -85,B 0,C 180,E1 6857.604,E2 6857.604} C_VEL
LIN {X 0,Y 264.264,Z 746.663,A -85,B 0,C 180,E1 6856.454,E2 6856.454} C_VEL
LIN {X 0,Y 270.187,Z 726.256,A -85,B 0,C 180,E1 6855.511,E2 6855.511} C_VEL
LIN {X 0,Y 274.82,Z 704.253,A -85,B 0,C 180,E1 6854.738,E2 6854.738} C_VEL
LIN {X 0,Y 277.814,Z 681.776,A -85,B 0,C 180,E1 6854.161,E2 6854.161} C_VEL
LIN {X 0,Y 287.635,Z 590.013,A -85,B 0,C 180,E1 6852.503,E2 6852.503} C_VEL
LIN {X 0,Y 286.421,Z 587.512,A -85,B 0,C 180,E1 6850.459,E2 6850.459} C_VEL
LIN {X 0,Y 285.146,Z 584.762,A -85,B 0,C 180,E1 6847.252,E2 6847.252} C_VEL
LIN {X 0,Y 284.449,Z 584.42,A -85,B 0,C 180,E1 6843.225,E2 6843.225} C_VEL
LIN {X 0,Y 284.465,Z 585.002,A -85,B 0,C 180,E1 6841.612,E2 6841.612} C_VEL
LIN {X 0,Y 285.119,Z 588.168,A -85,B 0,C 180,E1 6837.991,E2 6837.991} C_VEL
LIN {X 0,Y 286.4,Z 592.477,A -85,B 0,C 180,E1 6834.893,E2 6834.893} C_VEL
LIN {X 0,Y 287.531,Z 596.416,A -85,B 0,C 180,E1 6832.883,E2 6832.883} C_VEL
LIN {X 0,Y 274.666,Z 711.56,A -85,B 0,C 180,E1 6830.811,E2 6830.811} C_VEL
LIN {X 0,Y 270.847,Z 731.539,A -85,B 0,C 180,E1 6830.36,E2 6830.36} C_VEL
LIN {X 0,Y 268.519,Z 740.095,A -85,B 0,C 180,E1 6830.413,E2 6830.413} C_VEL
LIN {X 0,Y 261.992,Z 757.689,A -85,B 0,C 180,E1 6831.123,E2 6831.123} C_VEL
LIN {X 0,Y 259.222,Z 764.93,A -85,B 0,C 180,E1 6831.095,E2 6831.095} C_VEL
LIN {X 0,Y 251.001,Z 785.33,A -85,B 0,C 180,E1 6830.342,E2 6830.342} C_VEL
LIN {X 0,Y 241.584,Z 804.696,A -85,B 0,C 180,E1 6829.38,E2 6829.38} C_VEL
LIN {X 0,Y 230.893,Z 823.277,A -85,B 0,C 180,E1 6828.122,E2 6828.122} C_VEL
LIN {X 0,Y 218.625,Z 841.799,A -85,B 0,C 180,E1 6826.429,E2 6826.429} C_VEL
LIN {X 0,Y 205.62,Z 859.017,A -85,B 0,C 180,E1 6824.307,E2 6824.307} C_VEL
LIN {X 0,Y 191.772,Z 875.292,A -85,B 0,C 180,E1 6821.592,E2 6821.592} C_VEL
LIN {X 0,Y 177.686,Z 890.076,A -85,B 0,C 180,E1 6818.187,E2 6818.187} C_VEL
LIN {X 0,Y 163.643,Z 903.526,A -85,B 0,C 180,E1 6813.902,E2 6813.902} C_VEL
LIN {X 0,Y 149.428,Z 916.227,A -85,B 0,C 180,E1 6808.182,E2 6808.182} C_VEL
LIN {X 0,Y 137.033,Z 926.87,A -85,B 0,C 180,E1 6801.322,E2 6801.322} C_VEL
LIN {X 0,Y 126.527,Z 936.045,A -85,B 0,C 180,E1 6792.809,E2 6792.809} C_VEL
LIN {X 0,Y 119.034,Z 943.343,A -85,B 0,C 180,E1 6782.864,E2 6782.864} C_VEL
LIN {X 0,Y 115.225,Z 948.6,A -85,B 0,C 180,E1 6772.445,E2 6772.445} C_VEL
LIN {X 0,Y 114.612,Z 952.099,A -85,B 0,C 180,E1 6762.086,E2 6762.086} C_VEL
LIN {X 0,Y 115.716,Z 953.561,A -85,B 0,C 180,E1 6753.965,E2 6753.965} C_VEL
LIN {X 0,Y 116.165,Z 953.84,A -85,B 0,C 180,E1 6749.509,E2 6749.509} C_VEL
LIN {X 0,Y 115.362,Z 953.346,A -85,B 0,C 180,E1 6744.032,E2 6744.032} C_VEL
LIN {X 0,Y 114.518,Z 951.174,A -85,B 0,C 180,E1 6734.819,E2 6734.819} C_VEL
LIN {X 0,Y 115.981,Z 947.269,A -85,B 0,C 180,E1 6724.471,E2 6724.471} C_VEL
LIN {X 0,Y 120.909,Z 941.301,A -85,B 0,C 180,E1 6714.052,E2 6714.052} C_VEL
LIN {X 0,Y 129.234,Z 933.506,A -85,B 0,C 180,E1 6704.627,E2 6704.627} C_VEL
LIN {X 0,Y 140.52,Z 923.782,A -85,B 0,C 180,E1 6696.492,E2 6696.492} C_VEL
LIN {X 0,Y 152.964,Z 913.076,A -85,B 0,C 180,E1 6690.219,E2 6690.219} C_VEL
LIN {X 0,Y 166.673,Z 900.617,A -85,B 0,C 180,E1 6685.079,E2 6685.079} C_VEL
LIN {X 0,Y 180.203,Z 887.329,A -85,B 0,C 180,E1 6681.139,E2 6681.139} C_VEL
LIN {X 0,Y 194.746,Z 871.687,A -85,B 0,C 180,E1 6677.773,E2 6677.773} C_VEL
LIN {X 0,Y 208.254,Z 855.487,A -85,B 0,C 180,E1 6675.222,E2 6675.222} C_VEL
LIN {X 0,Y 221.268,Z 837.811,A -85,B 0,C 180,E1 6673.174,E2 6673.174} C_VEL
LIN {X 0,Y 232.726,Z 819.913,A -85,B 0,C 180,E1 6671.638,E2 6671.638} C_VEL
LIN {X 0,Y 243.358,Z 800.765,A -85,B 0,C 180,E1 6670.414,E2 6670.414} C_VEL
LIN {X 0,Y 252.409,Z 781.668,A -85,B 0,C 180,E1 6669.516,E2 6669.516} C_VEL
LIN {X 0,Y 260.489,Z 760.834,A -85,B 0,C 180,E1 6668.784,E2 6668.784} C_VEL
LIN {X 0,Y 266.891,Z 739.585,A -85,B 0,C 180,E1 6668.186,E2 6668.186} C_VEL
LIN {X 0,Y 271.802,Z 717.218,A -85,B 0,C 180,E1 6667.673,E2 6667.673} C_VEL
LIN {X 0,Y 275.29,Z 692.108,A -85,B 0,C 180,E1 6667.202,E2 6667.202} C_VEL
LIN {X 0,Y 285.386,Z 601.708,A -85,B 0,C 180,E1 6665.629,E2 6665.629} C_VEL
LIN {X 0,Y 284.185,Z 597.3,A -85,B 0,C 180,E1 6662.924,E2 6662.924} C_VEL
LIN {X 0,Y 283.532,Z 594.622,A -85,B 0,C 180,E1 6660.606,E2 6660.606} C_VEL
LIN {X 0,Y 283.235,Z 592.311,A -85,B 0,C 180,E1 6657.572,E2 6657.572} C_VEL
LIN {X 0,Y 283.742,Z 592.356,A -85,B 0,C 180,E1 6653.322,E2 6653.322} C_VEL
LIN {X 0,Y 284.246,Z 593.211,A -85,B 0,C 180,E1 6651.707,E2 6651.707} C_VEL
LIN {X 0,Y 285.533,Z 596.177,A -85,B 0,C 180,E1 6648.836,E2 6648.836} C_VEL
LIN {X 0,Y 275.406,Z 688.202,A -85,B 0,C 180,E1 6647.232,E2 6647.232} C_VEL
LIN {X 0,Y 272.151,Z 709.916,A -85,B 0,C 180,E1 6646.648,E2 6646.648} C_VEL
LIN {X 0,Y 267.245,Z 730.992,A -85,B 0,C 180,E1 6645.888,E2 6645.888} C_VEL
LIN {X 0,Y 261.338,Z 750.016,A -85,B 0,C 180,E1 6645.001,E2 6645.001} C_VEL
LIN {X 0,Y 253.906,Z 769.156,A -85,B 0,C 180,E1 6643.891,E2 6643.891} C_VEL
LIN {X 0,Y 245.22,Z 787.484,A -85,B 0,C 180,E1 6642.554,E2 6642.554} C_VEL
LIN {X 0,Y 235.325,Z 804.895,A -85,B 0,C 180,E1 6640.954,E2 6640.954} C_VEL
LIN {X 0,Y 223.9,Z 822.108,A -85,B 0,C 180,E1 6638.941,E2 6638.941} C_VEL
LIN {X 0,Y 212.307,Z 837.249,A -85,B 0,C 180,E1 6636.67,E2 6636.67} C_VEL
LIN {X 0,Y 199.429,Z 851.933,A -85,B 0,C 180,E1 6633.809,E2 6633.809} C_VEL
LIN {X 0,Y 186.236,Z 865.026,A -85,B 0,C 180,E1 6630.4,E2 6630.4} C_VEL
LIN {X 0,Y 173.036,Z 876.644,A -85,B 0,C 180,E1 6626.302,E2 6626.302} C_VEL
LIN {X 0,Y 159.402,Z 887.329,A -85,B 0,C 180,E1 6621.05,E2 6621.05} C_VEL
LIN {X 0,Y 147.179,Z 895.967,A -85,B 0,C 180,E1 6614.945,E2 6614.945} C_VEL
LIN {X 0,Y 136.654,Z 902.807,A -85,B 0,C 180,E1 6607.917,E2 6607.917} C_VEL
LIN {X 0,Y 127.805,Z 908.106,A -85,B 0,C 180,E1 6599.524,E2 6599.524} C_VEL
LIN {X 0,Y 121.529,Z 911.753,A -85,B 0,C 180,E1 6590.211,E2 6590.211} C_VEL
LIN {X 0,Y 117.942,Z 913.892,A -85,B 0,C 180,E1 6580.252,E2 6580.252} C_VEL
LIN {X 0,Y 116.838,Z 914.593,A -85,B 0,C 180,E1 6570.979,E2 6570.979} C_VEL
LIN {X 0,Y 117.622,Z 914.088,A -85,B 0,C 180,E1 6561.198,E2 6561.198} C_VEL
LIN {X 0,Y 120.836,Z 912.23,A -85,B 0,C 180,E1 6551.174,E2 6551.174} C_VEL
LIN {X 0,Y 127.049,Z 908.654,A -85,B 0,C 180,E1 6541.312,E2 6541.312} C_VEL
LIN {X 0,Y 136.111,Z 903.201,A -85,B 0,C 180,E1 6532.434,E2 6532.434} C_VEL
LIN {X 0,Y 146.534,Z 896.492,A -85,B 0,C 180,E1 6525.351,E2 6525.351} C_VEL
LIN {X 0,Y 158.676,Z 887.999,A -85,B 0,C 180,E1 6519.195,E2 6519.195} C_VEL
LIN {X 0,Y 171.539,Z 878.063,A -85,B 0,C 180,E1 6514.145,E2 6514.145} C_VEL
LIN {X 0,Y 184.67,Z 866.722,A -85,B 0,C 180,E1 6509.978,E2 6509.978} C_VEL
LIN {X 0,Y 197.76,Z 853.85,A -85,B 0,C 180,E1 6506.514,E2 6506.514} C_VEL
LIN {X 0,Y 210.592,Z 839.542,A -85,B 0,C 180,E1 6503.615,E2 6503.615} C_VEL
LIN {X 0,Y 222.986,Z 823.702,A -85,B 0,C 180,E1 6501.159,E2 6501.159} C_VEL
LIN {X 0,Y 233.976,Z 807.522,A -85,B 0,C 180,E1 6499.208,E2 6499.208} C_VEL
LIN {X 0,Y 244.283,Z 789.684,A -85,B 0,C 180,E1 6497.524,E2 6497.524} C_VEL
LIN {X 0,Y 252.963,Z 771.783,A -85,B 0,C 180,E1 6496.179,E2 6496.179} C_VEL
LIN {X 0,Y 260.837,Z 752.122,A -85,B 0,C 180,E1 6495.006,E2 6495.006} C_VEL
LIN {X 0,Y 267.2,Z 732.079,A -85,B 0,C 180,E1 6494.056,E2 6494.056} C_VEL
LIN {X 0,Y 272.219,Z 710.782,A -85,B 0,C 180,E1 6493.28,E2 6493.28} C_VEL
LIN {X 0,Y 275.489,Z 689.435,A -85,B 0,C 180,E1 6492.699,E2 6492.699} C_VEL
LIN {X 0,Y 283.934,Z 612.759,A -85,B 0,C 180,E1 6491.338,E2 6491.338} C_VEL
LIN {X 0,Y 285.759,Z 596.162,A -85,B 0,C 180,E1 6491.045,E2 6491.045} C_VEL
LIN {X 0,Y 284.113,Z 592.665,A -85,B 0,C 180,E1 6487.076,E2 6487.076} C_VEL
LIN {X 0,Y 283.471,Z 592.388,A -85,B 0,C 180,E1 6483.033,E2 6483.033} C_VEL
LIN {X 0,Y 283.478,Z 593.047,A -85,B 0,C 180,E1 6481.617,E2 6481.617} C_VEL
LIN {X 0,Y 284.019,Z 595.972,A -85,B 0,C 180,E1 6478.286,E2 6478.286} C_VEL
LIN {X 0,Y 285.171,Z 600.157,A -85,B 0,C 180,E1 6475.274,E2 6475.274} C_VEL
LIN {X 0,Y 285.585,Z 602.088,A -85,B 0,C 180,E1 6474.368,E2 6474.368} C_VEL
LIN {X 0,Y 273.198,Z 710.614,A -85,B 0,C 180,E1 6472.472,E2 6472.472} C_VEL
LIN {X 0,Y 268.811,Z 732.846,A -85,B 0,C 180,E1 6471.99,E2 6471.99} C_VEL
LIN {X 0,Y 262.877,Z 754.175,A -85,B 0,C 180,E1 6471.427,E2 6471.427} C_VEL
LIN {X 0,Y 259.222,Z 764.93,A -85,B 0,C 180,E1 6471.095,E2 6471.095} C_VEL
LIN {X 0,Y 256.286,Z 772.2,A -85,B 0,C 180,E1 6471.068,E2 6471.068} C_VEL
LIN {X 0,Y 247.146,Z 789.883,A -85,B 0,C 180,E1 6471.716,E2 6471.716} C_VEL
LIN {X 0,Y 243.515,Z 796.677,A -85,B 0,C 180,E1 6471.629,E2 6471.629} C_VEL
LIN {X 0,Y 233.103,Z 815.665,A -85,B 0,C 180,E1 6470.562,E2 6470.562} C_VEL
LIN {X 0,Y 220.934,Z 834.575,A -85,B 0,C 180,E1 6469.103,E2 6469.103} C_VEL
LIN {X 0,Y 208.055,Z 851.913,A -85,B 0,C 180,E1 6467.287,E2 6467.287} C_VEL
LIN {X 0,Y 193.694,Z 868.948,A -85,B 0,C 180,E1 6464.845,E2 6464.845} C_VEL
LIN {X 0,Y 179.797,Z 883.654,A -85,B 0,C 180,E1 6461.964,E2 6461.964} C_VEL
LIN {X 0,Y 164.896,Z 897.899,A -85,B 0,C 180,E1 6458.072,E2 6458.072} C_VEL
LIN {X 0,Y 150.087,Z 910.72,A -85,B 0,C 180,E1 6453.064,E2 6453.064} C_VEL
LIN {X 0,Y 136.314,Z 921.921,A -85,B 0,C 180,E1 6446.733,E2 6446.733} C_VEL
LIN {X 0,Y 123.972,Z 931.732,A -85,B 0,C 180,E1 6438.592,E2 6438.592} C_VEL
LIN {X 0,Y 114.575,Z 939.615,A -85,B 0,C 180,E1 6428.924,E2 6428.924} C_VEL
LIN {X 0,Y 108.705,Z 945.642,A -85,B 0,C 180,E1 6417.974,E2 6417.974} C_VEL
LIN {X 0,Y 106.625,Z 949.65,A -85,B 0,C 180,E1 6406.9,E2 6406.9} C_VEL
LIN {X 0,Y 107.278,Z 951.919,A -85,B 0,C 180,E1 6396.96,E2 6396.96} C_VEL
LIN {X 0,Y 108.267,Z 952.515,A -85,B 0,C 180,E1 6390.531,E2 6390.531} C_VEL
LIN {X 0,Y 107.735,Z 952.21,A -85,B 0,C 180,E1 6385.744,E2 6385.744} C_VEL
LIN {X 0,Y 106.621,Z 950.709,A -85,B 0,C 180,E1 6376.997,E2 6376.997} C_VEL
LIN {X 0,Y 107.59,Z 947.169,A -85,B 0,C 180,E1 6365.869,E2 6365.869} C_VEL
LIN {X 0,Y 112.197,Z 941.76,A -85,B 0,C 180,E1 6354.608,E2 6354.608} C_VEL
LIN {X 0,Y 120.465,Z 934.562,A -85,B 0,C 180,E1 6344.464,E2 6344.464} C_VEL
LIN {X 0,Y 132.23,Z 925.114,A -85,B 0,C 180,E1 6335.607,E2 6335.607} C_VEL
LIN {X 0,Y 145.14,Z 914.693,A -85,B 0,C 180,E1 6328.981,E2 6328.981} C_VEL
LIN {X 0,Y 160.112,Z 901.958,A -85,B 0,C 180,E1 6323.384,E2 6323.384} C_VEL
LIN {X 0,Y 174.727,Z 888.471,A -85,B 0,C 180,E1 6319.251,E2 6319.251} C_VEL
LIN {X 0,Y 189.288,Z 873.662,A -85,B 0,C 180,E1 6316.004,E2 6316.004} C_VEL
LIN {X 0,Y 203.514,Z 857.335,A -85,B 0,C 180,E1 6313.43,E2 6313.43} C_VEL
LIN {X 0,Y 216.294,Z 840.763,A -85,B 0,C 180,E1 6311.509,E2 6311.509} C_VEL
LIN {X 0,Y 228.858,Z 822.178,A -85,B 0,C 180,E1 6309.912,E2 6309.912} C_VEL
LIN {X 0,Y 239.722,Z 803.62,A -85,B 0,C 180,E1 6308.739,E2 6308.739} C_VEL
LIN {X 0,Y 249.465,Z 783.842,A -85,B 0,C 180,E1 6307.832,E2 6307.832} C_VEL
LIN {X 0,Y 257.445,Z 764.273,A -85,B 0,C 180,E1 6307.164,E2 6307.164} C_VEL
LIN {X 0,Y 264.481,Z 742.571,A -85,B 0,C 180,E1 6306.568,E2 6306.568} C_VEL
LIN {X 0,Y 269.698,Z 720.925,A -85,B 0,C 180,E1 6306.08,E2 6306.08} C_VEL
LIN {X 0,Y 273.262,Z 698.333,A -85,B 0,C 180,E1 6305.658,E2 6305.658} C_VEL
LIN {X 0,Y 283.621,Z 607.276,A -85,B 0,C 180,E1 6304.093,E2 6304.093} C_VEL
LIN {X 0,Y 282.585,Z 602.812,A -85,B 0,C 180,E1 6300.81,E2 6300.81} C_VEL
LIN {X 0,Y 282.243,Z 600.213,A -85,B 0,C 180,E1 6297.294,E2 6297.294} C_VEL
LIN {X 0,Y 282.776,Z 600.311,A -85,B 0,C 180,E1 6293.299,E2 6293.299} C_VEL
LIN {X 0,Y 283.27,Z 601.299,A -85,B 0,C 180,E1 6291.679,E2 6291.679} C_VEL
LIN {X 0,Y 283.773,Z 602.8,A -85,B 0,C 180,E1 6290.33,E2 6290.33} C_VEL
LIN {X 0,Y 274.061,Z 689.085,A -85,B 0,C 180,E1 6288.867,E2 6288.867} C_VEL
LIN {X 0,Y 270.716,Z 710.877,A -85,B 0,C 180,E1 6288.297,E2 6288.297} C_VEL
LIN {X 0,Y 265.701,Z 731.997,A -85,B 0,C 180,E1 6287.562,E2 6287.562} C_VEL
LIN {X 0,Y 259.422,Z 751.743,A -85,B 0,C 180,E1 6286.673,E2 6286.673} C_VEL
LIN {X 0,Y 251.842,Z 770.743,A -85,B 0,C 180,E1 6285.607,E2 6285.607} C_VEL
LIN {X 0,Y 242.692,Z 789.574,A -85,B 0,C 180,E1 6284.277,E2 6284.277} C_VEL
LIN {X 0,Y 232.008,Z 807.779,A -85,B 0,C 180,E1 6282.643,E2 6282.643} C_VEL
LIN {X 0,Y 220.764,Z 824.114,A -85,B 0,C 180,E1 6280.77,E2 6280.77} C_VEL
LIN {X 0,Y 208.469,Z 839.605,A -85,B 0,C 180,E1 6278.49,E2 6278.49} C_VEL
LIN {X 0,Y 196.07,Z 853.306,A -85,B 0,C 180,E1 6275.881,E2 6275.881} C_VEL
LIN {X 0,Y 182.478,Z 866.37,A -85,B 0,C 180,E1 6272.566,E2 6272.566} C_VEL
LIN {X 0,Y 168.769,Z 877.995,A -85,B 0,C 180,E1 6268.541,E2 6268.541} C_VEL
LIN {X 0,Y 154.538,Z 888.676,A -85,B 0,C 180,E1 6263.338,E2 6263.338} C_VEL
LIN {X 0,Y 141.671,Z 897.307,A -85,B 0,C 180,E1 6257.214,E2 6257.214} C_VEL
LIN {X 0,Y 130.113,Z 904.35,A -85,B 0,C 180,E1 6249.783,E2 6249.783} C_VEL
LIN {X 0,Y 120.576,Z 909.671,A -85,B 0,C 180,E1 6240.934,E2 6240.934} C_VEL
LIN {X 0,Y 113.874,Z 913.224,A -85,B 0,C 180,E1 6231.096,E2 6231.096} C_VEL
LIN {X 0,Y 110.055,Z 915.278,A -85,B 0,C 180,E1 6220.466,E2 6220.466} C_VEL
LIN {X 0,Y 108.944,Z 915.962,A -85,B 0,C 180,E1 6209.998,E2 6209.998} C_VEL
LIN {X 0,Y 110.039,Z 915.305,A -85,B 0,C 180,E1 6199.529,E2 6199.529} C_VEL
LIN {X 0,Y 114.092,Z 913.151,A -85,B 0,C 180,E1 6188.404,E2 6188.404} C_VEL
LIN {X 0,Y 120.915,Z 909.539,A -85,B 0,C 180,E1 6178.605,E2 6178.605} C_VEL
LIN {X 0,Y 130.416,Z 904.264,A -85,B 0,C 180,E1 6169.912,E2 6169.912} C_VEL
LIN {X 0,Y 142.209,Z 897.087,A -85,B 0,C 180,E1 6162.422,E2 6162.422} C_VEL
LIN {X 0,Y 154.941,Z 888.526,A -85,B 0,C 180,E1 6156.42,E2 6156.42} C_VEL
LIN {X 0,Y 168.691,Z 878.222,A -85,B 0,C 180,E1 6151.412,E2 6151.412} C_VEL
LIN {X 0,Y 182.401,Z 866.643,A -85,B 0,C 180,E1 6147.382,E2 6147.382} C_VEL
LIN {X 0,Y 195.993,Z 853.607,A -85,B 0,C 180,E1 6144.063,E2 6144.063} C_VEL
LIN {X 0,Y 209.233,Z 838.991,A -85,B 0,C 180,E1 6141.288,E2 6141.288} C_VEL
LIN {X 0,Y 221.55,Z 823.366,A -85,B 0,C 180,E1 6139.021,E2 6139.021} C_VEL
LIN {X 0,Y 233.246,Z 806.152,A -85,B 0,C 180,E1 6137.088,E2 6137.088} C_VEL
LIN {X 0,Y 243.359,Z 788.748,A -85,B 0,C 180,E1 6135.554,E2 6135.554} C_VEL
LIN {X 0,Y 252.227,Z 770.437,A -85,B 0,C 180,E1 6134.27,E2 6134.27} C_VEL
LIN {X 0,Y 259.812,Z 751.333,A -85,B 0,C 180,E1 6133.205,E2 6133.205} C_VEL
LIN {X 0,Y 266.401,Z 730.252,A -85,B 0,C 180,E1 6132.27,E2 6132.27} C_VEL
LIN {X 0,Y 271.194,Z 709.532,A -85,B 0,C 180,E1 6131.565,E2 6131.565} C_VEL
LIN {X 0,Y 274.499,Z 687.624,A -85,B 0,C 180,E1 6131.002,E2 6131.002} C_VEL
LIN {X 0,Y 283.991,Z 602.759,A -85,B 0,C 180,E1 6129.525,E2 6129.525} C_VEL
LIN {X 0,Y 283.083,Z 600.568,A -85,B 0,C 180,E1 6126.898,E2 6126.898} C_VEL
LIN {X 0,Y 282.497,Z 600.33,A -85,B 0,C 180,E1 6123.044,E2 6123.044} C_VEL
LIN {X 0,Y 282.491,Z 601.088,A -85,B 0,C 180,E1 6121.623,E2 6121.623} C_VEL
LIN {X 0,Y 282.931,Z 603.778,A -85,B 0,C 180,E1 6118.583,E2 6118.583} C_VEL
LIN {X 0,Y 283.852,Z 607.521,A -85,B 0,C 180,E1 6115.876,E2 6115.876} C_VEL
LIN {X 0,Y 271.979,Z 709.563,A -85,B 0,C 180,E1 6114.152,E2 6114.152} C_VEL
LIN {X 0,Y 267.508,Z 731.898,A -85,B 0,C 180,E1 6113.693,E2 6113.693} C_VEL
LIN {X 0,Y 261.546,Z 753.046,A -85,B 0,C 180,E1 6113.17,E2 6113.17} C_VEL
LIN {X 0,Y 253.468,Z 775.039,A -85,B 0,C 180,E1 6112.503,E2 6112.503} C_VEL
LIN {X 0,Y 244.494,Z 794.787,A -85,B 0,C 180,E1 6111.719,E2 6111.719} C_VEL
LIN {X 0,Y 243.515,Z 796.677,A -85,B 0,C 180,E1 6111.629,E2 6111.629} C_VEL
LIN {X 0,Y 239.704,Z 803.576,A -85,B 0,C 180,E1 6111.513,E2 6111.513} C_VEL
LIN {X 0,Y 228.509,Z 820.055,A -85,B 0,C 180,E1 6111.949,E2 6111.949} C_VEL
LIN {X 0,Y 224.103,Z 826.369,A -85,B 0,C 180,E1 6111.742,E2 6111.742} C_VEL
LIN {X 0,Y 211.277,Z 844.329,A -85,B 0,C 180,E1 6110.191,E2 6110.191} C_VEL
LIN {X 0,Y 197.746,Z 860.754,A -85,B 0,C 180,E1 6108.244,E2 6108.244} C_VEL
LIN {X 0,Y 183.582,Z 876.013,A -85,B 0,C 180,E1 6105.785,E2 6105.785} C_VEL
LIN {X 0,Y 168.707,Z 890.382,A -85,B 0,C 180,E1 6102.574,E2 6102.574} C_VEL
LIN {X 0,Y 152.908,Z 904.11,A -85,B 0,C 180,E1 6098.196,E2 6098.196} C_VEL
LIN {X 0,Y 137.552,Z 916.243,A -85,B 0,C 180,E1 6092.468,E2 6092.468} C_VEL
LIN {X 0,Y 123.942,Z 926.349,A -85,B 0,C 180,E1 6085.366,E2 6085.366} C_VEL
LIN {X 0,Y 112.195,Z 935.028,A -85,B 0,C 180,E1 6076.204,E2 6076.204} C_VEL
LIN {X 0,Y 103.803,Z 941.862,A -85,B 0,C 180,E1 6065.304,E2 6065.304} C_VEL
LIN {X 0,Y 99.485,Z 946.654,A -85,B 0,C 180,E1 6053.704,E2 6053.704} C_VEL
LIN {X 0,Y 98.794,Z 949.797,A -85,B 0,C 180,E1 6041.679,E2 6041.679} C_VEL
LIN {X 0,Y 99.944,Z 950.969,A -85,B 0,C 180,E1 6033.443,E2 6033.443} C_VEL
LIN {X 0,Y 100.365,Z 951.18,A -85,B 0,C 180,E1 6029.431,E2 6029.431} C_VEL
LIN {X 0,Y 99.184,Z 950.441,A -85,B 0,C 180,E1 6021.89,E2 6021.89} C_VEL
LIN {X 0,Y 98.803,Z 948.074,A -85,B 0,C 180,E1 6011.109,E2 6011.109} C_VEL
LIN {X 0,Y 102.121,Z 943.406,A -85,B 0,C 180,E1 5998.088,E2 5998.088} C_VEL
LIN {X 0,Y 109.423,Z 937.151,A -85,B 0,C 180,E1 5986.748,E2 5986.748} C_VEL
LIN {X 0,Y 120.287,Z 928.997,A -85,B 0,C 180,E1 5977.073,E2 5977.073} C_VEL
LIN {X 0,Y 133.247,Z 919.357,A -85,B 0,C 180,E1 5969.503,E2 5969.503} C_VEL
LIN {X 0,Y 148.139,Z 907.798,A -85,B 0,C 180,E1 5963.392,E2 5963.392} C_VEL
LIN {X 0,Y 162.766,Z 895.553,A -85,B 0,C 180,E1 5958.934,E2 5958.934} C_VEL
LIN {X 0,Y 178.248,Z 881.22,A -85,B 0,C 180,E1 5955.271,E2 5955.271} C_VEL
LIN {X 0,Y 193.036,Z 865.821,A -85,B 0,C 180,E1 5952.512,E2 5952.512} C_VEL
LIN {X 0,Y 206.966,Z 849.455,A -85,B 0,C 180,E1 5950.379,E2 5950.379} C_VEL
LIN {X 0,Y 220.162,Z 831.81,A -85,B 0,C 180,E1 5948.699,E2 5948.699} C_VEL
LIN {X 0,Y 231.891,Z 813.79,A -85,B 0,C 180,E1 5947.432,E2 5947.432} C_VEL
LIN {X 0,Y 242.474,Z 794.624,A -85,B 0,C 180,E1 5946.453,E2 5946.453} C_VEL
LIN {X 0,Y 251.739,Z 774.67,A -85,B 0,C 180,E1 5945.719,E2 5945.719} C_VEL
LIN {X 0,Y 259.719,Z 753.471,A -85,B 0,C 180,E1 5945.118,E2 5945.118} C_VEL
LIN {X 0,Y 265.952,Z 732.034,A -85,B 0,C 180,E1 5944.619,E2 5944.619} C_VEL
LIN {X 0,Y 270.549,Z 709.662,A -85,B 0,C 180,E1 5944.184,E2 5944.184} C_VEL
LIN {X 0,Y 276.955,Z 657.122,A -85,B 0,C 180,E1 5943.312,E2 5943.312} C_VEL
LIN {X 0,Y 282.047,Z 613.204,A -85,B 0,C 180,E1 5942.59,E2 5942.59} C_VEL
LIN {X 0,Y 281.43,Z 610.208,A -85,B 0,C 180,E1 5940,E2 5940} C_VEL
LIN {X 0,Y 281.267,Z 608.136,A -85,B 0,C 180,E1 5937.147,E2 5937.147} C_VEL
LIN {X 0,Y 281.817,Z 608.266,A -85,B 0,C 180,E1 5933.276,E2 5933.276} C_VEL
LIN {X 0,Y 282.233,Z 609.211,A -85,B 0,C 180,E1 5931.846,E2 5931.846} C_VEL
LIN {X 0,Y 272.913,Z 690.174,A -85,B 0,C 180,E1 5930.512,E2 5930.512} C_VEL
LIN {X 0,Y 269.474,Z 712.017,A -85,B 0,C 180,E1 5929.956,E2 5929.956} C_VEL
LIN {X 0,Y 264.326,Z 733.221,A -85,B 0,C 180,E1 5929.246,E2 5929.246} C_VEL
LIN {X 0,Y 257.909,Z 752.976,A -85,B 0,C 180,E1 5928.391,E2 5928.391} C_VEL
LIN {X 0,Y 250.007,Z 772.33,A -85,B 0,C 180,E1 5927.349,E2 5927.349} C_VEL
LIN {X 0,Y 240.978,Z 790.55,A -85,B 0,C 180,E1 5926.119,E2 5926.119} C_VEL
LIN {X 0,Y 230.228,Z 808.539,A -85,B 0,C 180,E1 5924.582,E2 5924.582} C_VEL
LIN {X 0,Y 218.734,Z 824.951,A -85,B 0,C 180,E1 5922.794,E2 5922.794} C_VEL
LIN {X 0,Y 205.706,Z 840.996,A -85,B 0,C 180,E1 5920.535,E2 5920.535} C_VEL
LIN {X 0,Y 192.977,Z 854.677,A -85,B 0,C 180,E1 5918.022,E2 5918.022} C_VEL
LIN {X 0,Y 178.97,Z 867.734,A -85,B 0,C 180,E1 5914.815,E2 5914.815} C_VEL
LIN {X 0,Y 164.773,Z 879.346,A -85,B 0,C 180,E1 5910.891,E2 5910.891} C_VEL
LIN {X 0,Y 149.936,Z 890.019,A -85,B 0,C 180,E1 5905.771,E2 5905.771} C_VEL
LIN {X 0,Y 136.403,Z 898.648,A -85,B 0,C 180,E1 5899.661,E2 5899.661} C_VEL
LIN {X 0,Y 124.298,Z 905.595,A -85,B 0,C 180,E1 5892.262,E2 5892.262} C_VEL
LIN {X 0,Y 113.843,Z 911.008,A -85,B 0,C 180,E1 5882.987,E2 5882.987} C_VEL
LIN {X 0,Y 106.517,Z 914.56,A -85,B 0,C 180,E1 5872.631,E2 5872.631} C_VEL
LIN {X 0,Y 102.295,Z 916.608,A -85,B 0,C 180,E1 5861.27,E2 5861.27} C_VEL
LIN {X 0,Y 101.055,Z 917.29,A -85,B 0,C 180,E1 5849.998,E2 5849.998} C_VEL
LIN {X 0,Y 102.279,Z 916.635,A -85,B 0,C 180,E1 5838.724,E2 5838.724} C_VEL
LIN {X 0,Y 106.76,Z 914.484,A -85,B 0,C 180,E1 5826.837,E2 5826.837} C_VEL
LIN {X 0,Y 114.215,Z 910.875,A -85,B 0,C 180,E1 5816.531,E2 5816.531} C_VEL
LIN {X 0,Y 124.444,Z 905.6,A -85,B 0,C 180,E1 5807.556,E2 5807.556} C_VEL
LIN {X 0,Y 136.985,Z 898.421,A -85,B 0,C 180,E1 5799.966,E2 5799.966} C_VEL
LIN {X 0,Y 150.591,Z 889.72,A -85,B 0,C 180,E1 5793.9,E2 5793.9} C_VEL
LIN {X 0,Y 165.469,Z 878.976,A -85,B 0,C 180,E1 5788.824,E2 5788.824} C_VEL
LIN {X 0,Y 179.706,Z 867.275,A -85,B 0,C 180,E1 5784.928,E2 5784.928} C_VEL
LIN {X 0,Y 193.745,Z 854.138,A -85,B 0,C 180,E1 5781.744,E2 5781.744} C_VEL
LIN {X 0,Y 207.361,Z 839.407,A -85,B 0,C 180,E1 5779.091,E2 5779.091} C_VEL
LIN {X 0,Y 219.548,Z 824.196,A -85,B 0,C 180,E1 5777.002,E2 5777.002} C_VEL
LIN {X 0,Y 231.503,Z 806.903,A -85,B 0,C 180,E1 5775.157,E2 5775.157} C_VEL
LIN {X 0,Y 241.82,Z 789.406,A -85,B 0,C 180,E1 5773.694,E2 5773.694} C_VEL
LIN {X 0,Y 250.863,Z 771.037,A -85,B 0,C 180,E1 5772.47,E2 5772.47} C_VEL
LIN {X 0,Y 258.59,Z 751.793,A -85,B 0,C 180,E1 5771.452,E2 5771.452} C_VEL
LIN {X 0,Y 265.304,Z 730.503,A -85,B 0,C 180,E1 5770.555,E2 5770.555} C_VEL
LIN {X 0,Y 270.161,Z 709.569,A -85,B 0,C 180,E1 5769.876,E2 5769.876} C_VEL
LIN {X 0,Y 273.456,Z 687.908,A -85,B 0,C 180,E1 5769.342,E2 5769.342} C_VEL
LIN {X 0,Y 282.441,Z 609.446,A -85,B 0,C 180,E1 5768.049,E2 5768.049} C_VEL
LIN {X 0,Y 282.004,Z 608.421,A -85,B 0,C 180,E1 5766.515,E2 5766.515} C_VEL
LIN {X 0,Y 281.523,Z 608.329,A -85,B 0,C 180,E1 5762.647,E2 5762.647} C_VEL
LIN {X 0,Y 281.84,Z 611.453,A -85,B 0,C 180,E1 5758.984,E2 5758.984} C_VEL
LIN {X 0,Y 282.246,Z 613.57,A -85,B 0,C 180,E1 5757.391,E2 5757.391} C_VEL
LIN {X 0,Y 270.964,Z 708.711,A -85,B 0,C 180,E1 5755.841,E2 5755.841} C_VEL
LIN {X 0,Y 266.419,Z 731.051,A -85,B 0,C 180,E1 5755.409,E2 5755.409} C_VEL
LIN {X 0,Y 260.561,Z 751.605,A -85,B 0,C 180,E1 5754.937,E2 5754.937} C_VEL
LIN {X 0,Y 252.624,Z 773.134,A -85,B 0,C 180,E1 5754.34,E2 5754.34} C_VEL
LIN {X 0,Y 243.452,Z 793.199,A -85,B 0,C 180,E1 5753.62,E2 5753.62} C_VEL
LIN {X 0,Y 232.858,Z 812.506,A -85,B 0,C 180,E1 5752.656,E2 5752.656} C_VEL
LIN {X 0,Y 224.103,Z 826.369,A -85,B 0,C 180,E1 5751.742,E2 5751.742} C_VEL
LIN {X 0,Y 219.522,Z 832.687,A -85,B 0,C 180,E1 5751.499,E2 5751.499} C_VEL
LIN {X 0,Y 206.385,Z 847.812,A -85,B 0,C 180,E1 5751.678,E2 5751.678} C_VEL
LIN {X 0,Y 201.298,Z 853.523,A -85,B 0,C 180,E1 5751.329,E2 5751.329} C_VEL
LIN {X 0,Y 186.31,Z 869.971,A -85,B 0,C 180,E1 5749.116,E2 5749.116} C_VEL
LIN {X 0,Y 170.833,Z 884.916,A -85,B 0,C 180,E1 5746.287,E2 5746.287} C_VEL
LIN {X 0,Y 155.069,Z 898.524,A -85,B 0,C 180,E1 5742.593,E2 5742.593} C_VEL
LIN {X 0,Y 139.337,Z 910.783,A -85,B 0,C 180,E1 5737.761,E2 5737.761} C_VEL
LIN {X 0,Y 124.197,Z 921.653,A -85,B 0,C 180,E1 5731.336,E2 5731.336} C_VEL
LIN {X 0,Y 110.173,Z 931.164,A -85,B 0,C 180,E1 5722.553,E2 5722.553} C_VEL
LIN {X 0,Y 99.802,Z 938.352,A -85,B 0,C 180,E1 5712.154,E2 5712.154} C_VEL
